Level_Manager();
_w1 := SEL(pump.Mode.eMode=eAnalog_Pump_Modes.Auto, pump.HMI_Volume_Target, pump.PLC_Volume_Target);
pump.Live_Rate := SEL(Pump.Config.Follow_ENABLE, _w1, Pump.Calibration_Rate* (pump.Config.Follow_Rate/100));
lcl_Target := _w1;
lcl_Seconds := SEL(pump.Mode.eMode=eAnalog_Pump_Modes.Auto, Pump.HMI_Volume_Target/PUMP.HMI_Rate_PCT, PUMP.PLC_Volume_Target/Pump.PLC_Rate_PCT);
_w2 := lcl_Target / ((PUMP.Config.Min_Speed/100.0) * (Pump.Calibration_Rate/60));
MAX_Time := _w2;
_w3 := lcl_Target / ((PUMP.Config.Max_Speed/100.0) * (Pump.Calibration_Rate/60));
Min_Time := _w3;
_w4 := SEL(lcl_Seconds<Min_time, SEL(lcl_Seconds>Max_Time, lcl_Seconds, _w2), _w3);
_w5 := REAL_TO_INT(_w4);
lcl_Seconds := _w5;
New_Pump_Time := _w5;
Base_PCT := SEL(lcl_Target=0, (Min_Time / _w4) * PUMP.Config.Max_Speed, 0.0);
_w6 := (Pump.Mode.eMode=eAnalog_Pump_Modes.Manual) OR Pump.PLC_Run AND (pump.Mode.eMode=eAnalog_Pump_Modes.Auto);
RUN_REQ := _w6;
_w7 := INT_TO_TIME(PUMP.Config.SuckBack_Seconds) * 1000;
_w8 := INT_TO_Time(New_Pump_Time) * 1000;
TON_0(IN := _w6, PT := _w8); // TON
_w9 := Pump.PLC_Run AND (pump.Mode.eMode=eAnalog_Pump_Modes.Auto);
_w10 := _w6 AND NOT TON_0.Q AND NOT (lcl_Target=0) OR (pump.Mode.eMode=eAnalog_Pump_Modes.Prime) OR (pump.Mode.eMode=eAnalog_Pump_Modes.Calibrate) OR Pump.Config.Follow_ENABLE;
F_TRIG_2(CLK := _w10); // F_Trig
Pump.Pump_FWD := _w10;
TP_2(IN := F_TRIG_2.Q AND (PUMP.Config.SuckBack_Seconds>1), PT := t#3s); // TP
TON_1(IN := TP_2.Q, PT := T#2s); // TON
TP_0(IN := TON_1.Q, PT := _w7); // TP
Pump.Pump_REV := TP_0.Q;
RUN := _w10 OR TP_0.Q;
REV := TP_0.Q;
PUMP.Batch_ETA := SEL(lcl_Target=0, SEL(_w6, New_Pump_time, TIME_TO_INT((_w8 - TON_0.ET) / 1000)), 0);
Pump.PCT_Remain := SEL(Run_REQ, 0.0, (1 - Pump.Volume_Delivered / pump.Live_Rate) * 100);
F_TRIG_0(CLK := _w9); // F_trig
IF F_TRIG_0.Q THEN _w11 := 0; END_IF
lcl_Target := _w11;
R_TRIG_0(CLK := Pump.Pump_FWD); // R_trig
Pump.Volume_Delivered := SEL(R_TRIG_0.Q, ((Pump.Calibration_Rate/60) * (Base_PCT/100)) * TIME_TO_INT(TON_0.ET / 1000), 0.0);
SET_Status();
F_TRIG_1(CLK := pump.Mode.eMode=eAnalog_Pump_Modes.Calibrate); // F_trig
_w12 := SEL(REV, 0, Pump.Config.SuckBack_Speed);
_w13 := (pump.HMI_Volume_Target / ((Pump.HMI_Volume_Target/ Pump.HMI_Rate_PCT) / 60.0)) * (100 / (pump.Config.Max_Speed*0.75));
Cal_Value := _w13;
IF F_TRIG_1.Q AND NOT TP_1.Q THEN _w14 := _w13; END_IF
Pump.Calibration_Rate := _w14;
_w15 := SEL(Pump.Pump_FWD, _w12, SEL(Pump.Config.Follow_ENABLE, SEL(pump.Mode.eMode=eAnalog_Pump_Modes.Prime, SEL(pump.Mode.eMode=eAnalog_Pump_Modes.Calibrate, Base_PCT, pump.Config.Max_Speed*0.75), pump.Config.Max_Speed), Pump.Config.Follow_Rate));
Pump.Pump_CV := _w15;
Speed := _w15;

ACTION Set_Status:
Pump.Status.eStatus := SEL((Pump.Mode.eMode=eAnalog_Pump_Modes.Auto) AND NOT Pump.PUMP_FWD AND PUMP.PLC_Run, SEL((Pump.Mode.eMode=eAnalog_Pump_Modes.Auto) AND Pump.Pump_FWD AND Pump.PLC_Run, SEL(Pump.Mode.eMode=eAnalog_Pump_Modes.Manual, SEL(Pump.Mode.eMode=eAnalog_Pump_Modes.Disabled, eAnalog_Pump_Status.IDLE, eAnalog_Pump_Status.Disabled), eAnalog_Pump_Status.Manual), eAnalog_Pump_Status.Running), eAnalog_Pump_Status.Complete);
END_ACTION

END_FUNCTION_BLOCK

// Level_2_Controls/Condensate_Trap_UDFB
FUNCTION_BLOCK Condensate_Trap_UDFB
VAR_INPUT
	LSHH:Burkert.DI_DUT;
	LSH:Burkert.DI_DUT;
	LSL:Burkert.DI_DUT;
	LSLL:Burkert.DI_DUT;
	Valve_Ready:BOOL;
	Steam_Load:REAL:=0;
	Purge_Duration:TIME:=T#15S;
	V2:BOOL:=FALSE;
	
END_VAR
VAR_OUTPUT
	ACV:REAL;
END_VAR

VAR
	R_TRIG_0: R_Trig;
	Valve_Min: REAL;
	Valve_Max: REAL;
	TON_0: TON;
	TON_2: TON;
	
	Target_CMD:REAL;
	T_mid:REAL;
	old_T_mid:REAL;
	t_Ramp:REAL:=0;
	Ramp: RAMP_REAL;
	Static_Time:Ton;
	Purge_TP:TP;
	purgeCount:UINT:=0;
	PurgeCount_rTrig:r_Trig;
END_VAR
VAR_IN_OUT
	Trap:cCondensate_Trap;
END_VAR
VAR // added by the converter: edge detectors and wires of the graphical bodies
    _w1, _w2, _w5, _w6, _w7, _w8, _w9, _w10, _w11, _w12, _w13, _w16, _w17, _w18 : ANY;
    _w3, _w4, _w14 : BOOL;
    _w15 : REAL;
END_VAR

_w1 := (LSL.Status.eStatus=Di_Status.Liquid_Detected) OR (LSL.Status.eStatus=Di_Status.Liquid_Detected_Alarm);
_w2 := (LSH.Status.eStatus=Di_Status.Liquid_Detected) OR (LSH.Status.eStatus=Di_Status.Liquid_Detected_Alarm);
_w3 := True;
IF _w3 THEN Positions(); END_IF
_w4 := _w3;
IF _w4 THEN Purge(); END_IF
IF _w4 THEN Status(); END_IF
_w5 := (LSHH.Status.eStatus=Di_Status.Liquid_Detected_Alarm) OR (LSHH.Status.eStatus=Di_Status.Liquid_Detected);
_w6 := (LSLL.Status.eStatus=Di_Status.Liquid_Detected) OR (LSLL.Status.eStatus=Di_Status.Liquid_Detected_Alarm);
_w7 := _w1 AND _w6;
IF TON_0.Q THEN _w8 := ACV+1; END_IF
_w9 := SEL(_w6, 100, Trap.Min_Valve_Positions[1]);
Trap.READY := Valve_Ready;
_w10 := _w2 AND _w7;
_w11 := _w5 AND _w10;
_w12 := SEL(_w11, SEL(_w10, SEL(_w7, _w9, Trap.Min_Valve_Positions[2]), Trap.Min_Valve_Positions[3]), 100);
_w13 := SEL(_w11, SEL(_w10, SEL(_w7, SEL(_w6, 0, Trap.Min_Valve_Positions[0]), Trap.Min_Valve_Positions[1]), Trap.Min_Valve_Positions[2]), Trap.Min_Valve_Positions[3]);
_w14 := _w13 <= 1;
TON_0(IN := NOT _w14 AND NOT TON_0.Q, PT := T#1s); // TON
_w15 := SEL(V2, SEL(_w14, LIMIT(_w13, _w8, _w12), 0.0), Target_CMD);
ACV := _w15;
Trap.CV := _w15;

ACTION Positions:


CASE Trap.Status OF
	eCondensate_Status.IDLE:
		Valve_Min:=0;
		Valve_Max:=0.1;
	eCondensate_Status.Stage_1:
		Valve_Min:=0;
		Valve_Max:=Trap.Min_Valve_Positions[0];
	eCondensate_Status.Stage_2:
		Valve_Min:=Trap.Min_Valve_Positions[0];
		Valve_Max:=Trap.Min_Valve_Positions[1];
	eCondensate_Status.High_Warning:
		Valve_Min:=Trap.Min_Valve_Positions[1];
		Valve_Max:=Trap.Min_Valve_Positions[2];
	eCondensate_Status.Fault:
		Valve_Min:=Trap.Min_Valve_Positions[2];
		Valve_Max:=Trap.Min_Valve_Positions[3];
		
		eCondensate_Status.HIGH_Alarm:
		Valve_Min:=Trap.Min_Valve_Positions[2];
		Valve_Max:=Trap.Min_Valve_Positions[3];
		
	eCondensate_Status.Level_Switch_Fault:
		Valve_Min:=0;
		Valve_Max:=0.1;
			
	eCondensate_Status.Purge:
		Valve_Min:=Trap.Min_Valve_Positions[1];
		Valve_Max:=Trap.Min_Valve_Positions[1]+1;
		Trap.PLC_Purge:=FALSE;
		IF Trap.Purge.eMode=Burkert.eHOA_Modes.Manual THEN Trap.Purge.eMode:=Burkert.eHOA_Modes.Auto; END_IF;
	
END_CASE

t_mid:=fbMidPoint(High:=Valve_max,Low:=Valve_Min);
Static_Time(PT:=T#2M, 
	IN:= (	t_mid = Old_t_mid AND 
			Trap.CV<15 AND
			Steam_Load>75)
	);
	
IF t_mid > Old_t_mid THEN
	t_Ramp:=Valve_Max;
	Old_T_Mid:=t_Mid;
END_IF;

IF t_mid < Old_t_mid THEN
	t_Ramp:=Valve_Min;
	Old_T_Mid:=t_Mid;
END_IF;



Ramp(
	IN:= t_ramp, 
	ASCEND:= 2, 
	DESCEND:= 2, 
	TIMEBASE:= T#1S, 
	RESET:= FALSE );

IF Ramp.OUT<5  THEN
	Target_CMD:=0;
ELSE
	Target_CMD:=LIMIT (Valve_Min,Ramp.OUT,MIN(Valve_Max,100));
END_IF
END_ACTION

ACTION Purge:
Purge_TP(PT:=Purge_Duration);




CASE Trap.Purge.eMode OF
	Burkert.eHOA_Modes.Off:
		Purge_TP.IN:=FALSE;
	Burkert.eHOA_Modes.Manual:
		Purge_TP.IN:=TRUE;
	Burkert.eHOA_Modes.Auto:
		Purge_TP.IN:=Static_Time.Q OR Trap.PLC_Purge;
		Trap.PLC_Purge:=FALSE;
END_CASE

PurgeCount_rTrig(CLK:=Purge_TP.IN);
IF PurgeCount_rTrig.Q THEN PurgeCount:=PurgeCount+1;	END_IF;
END_ACTION

ACTION Status:
TON_2(IN := ACV>99, PT := T#30s); // TON
_w16 := (LSLL.Status.eStatus=Di_Status.Liquid_Detected) OR (LSLL.Status.eStatus=Di_Status.Liquid_Detected_Alarm);
_w17 := ((LSL.Status.eStatus=Di_Status.Liquid_Detected) OR (LSL.Status.eStatus=Di_Status.Liquid_Detected_Alarm)) AND _w16;
_w18 := ((LSH.Status.eStatus=Di_Status.Liquid_Detected) OR (LSH.Status.eStatus=Di_Status.Liquid_Detected_Alarm)) AND _w17;
Trap.Status := SEL(Purge_TP.Q AND NOT (Trap.Purge.eMode=Burkert.eHOA_Modes.Off), SEL(LSHH.Raw AND NOT LSH.Raw OR LSH.Raw AND NOT LSL.Raw OR LSL.Raw AND NOT LSLL.Raw, SEL(TON_2.Q, SEL(((LSHH.Status.eStatus=Di_Status.Liquid_Detected_Alarm) OR (LSHH.Status.eStatus=Di_Status.Liquid_Detected)) AND _w18, SEL(_w18, SEL(_w17, SEL(_w16, eCondensate_Status.IDLE, eCondensate_Status.Stage_1), eCondensate_Status.Stage_2), eCondensate_Status.High_Warning), eCondensate_Status.HIGH_Alarm), eCondensate_Status.Fault), eCondensate_Status.Level_Switch_Fault), eCondensate_Status.Purge);
END_ACTION

END_FUNCTION_BLOCK

// Level_2_Controls/DofMaster
FUNCTION_BLOCK DofMaster
VAR_INPUT
	Config:REFERENCE TO cDOF_Master;
	ALL_Lines_Ready:BOOL;
	
END_VAR
VAR_OUTPUT
END_VAR
VAR
	R_Trig_0:R_trig;
	Batch_CLK:TON;
	R_Trig_1:R_trig;
	
END_VAR

Config.StrBatch_Mode:=Burkert_OSCAT_BASIC.REPLACE_ALL(str:=TO_STRING(Config.Batch_Mode.eMode), src:='_' , rep:=' ' );
Config.StrBatch_Status:=Burkert_OSCAT_BASIC.REPLACE_ALL(str:=TO_STRING(Config.Batch_Status.eStatus), src:='_' , rep:=' ' );
Config.StrBatch_Task:= Burkert_OSCAT_BASIC.REPLACE_ALL(str:=TO_STRING(Config.Batch_Task.eTask), src:='_' , rep:=' ' );

Config.Batch_Target_ms:=TO_UDINT((Config.Batch_Volume/Config.Batch_Rate)*60*1000);
Config.Batch_Elapsed_ms:=TO_UDINT(Batch_CLK.ET);
Config.Batch_Remain_ms:=Config.Batch_Target_ms-Config.Batch_Elapsed_ms;

R_trig_1( CLK:=(Config.Batch_Mode.eMode=Burkert.eHOA_Modes.Manual));

Batch_CLK(IN:=Config.Batch_Task.eTask=eBatch_Task.Run,PT:=T#6H);
Config.Batch_CLK:=Batch_CLK.ET;

IF Config.Current_Batch_Rate >0 THEN
	Config.Batch_ETA_ms:=TO_UDINT(	((Config.Batch_Volume-Config.Current_Batch_Volume) / Config.Current_Batch_Rate)*(60*1000)	);
ELSE
	Config.Batch_ETA_ms:=0;
END_IF;

IF Config.Batch_Rate >0 THEN	
	Config.Batch_Target_ms:=TO_UDINT((Config.Batch_Volume/Config.Batch_Rate)*60*1000);
	Config.Batch_Remain:=TO_TIME(		(Config.Batch_Volume/Config.Batch_Rate)*60*1000)-Config.Batch_CLK;
ELSE
	Config.Batch_Remain:=T#0MS;
	Config.Batch_Target_ms:=0;
END_IF


IF Config.Batch_Volume>0 THEN
	Config.Current_Batch_PCT:=(Config.Current_Batch_Volume/Config.Batch_Volume)*100;
ELSE
	Config.Current_Batch_PCT:=0;
	Config.Batch_Status.eStatus:=eBatch_Status.Idle;
END_IF;


IF ALL_Lines_Ready THEN
	Config.Batch_Status.eStatus:=eBatch_Status.Ready;
	IF Config.Batch_Task.eTask=eBatch_task.Resume THEN Task_resume(); END_IF;
	IF Config.Current_Batch_Rate>0.5 THEN Config.Batch_Status.eStatus:=eBatch_Status.Active; END_IF;
	
	CASE Config.Batch_Mode.eMode OF
		Burkert.eHOA_Modes.Auto:
			IF Config.PLC_Run THEN 
				Config.Batch_Task.eTask:=eBatch_Task.Run; 
			ELSE
				Config.Batch_Task.eTask:=eBatch_Task.OFF;
			END_IF;
		Burkert.eHOA_Modes.Manual:  
			IF R_trig_1.q	THEN	Config.Batch_Task.eTask:=eBatch_Task.Run; END_IF;
	ELSE
		Config.Batch_Task.eTask:=eBatch_Task.OFF;
		Config.Batch_Status.eStatus:=eBatch_Status.Disabled;
		Config.PLC_Run:=FALSE;
	END_CASE
ELSE
	Config.Batch_Task.eTask:=eBatch_Task.OFF;
	Config.Batch_Status.eStatus:=eBatch_Status.Fault;
	Config.Batch_Mode.eMode:=Burkert.eHOA_Modes.Off;
END_IF;

IF Config.Current_Batch_PCT>=100.0 THEN Config.Batch_Status.eStatus:=eBatch_Status.Complete; END_IF;


R_Trig_0(CLK:=Config.Batch_Task.eTask=eBatch_task.Run);
IF R_Trig_0.Q THEN
	Config.MasterID:=Config.MasterID+1;
END_IF;

END_FUNCTION_BLOCK

// Level_2_Controls/Duplex_VFD
FUNCTION_BLOCK Duplex_VFD
VAR_INPUT
	VFD1:REFERENCE TO Burkert.VFD_Control;
	VFD2:REFERENCE TO Burkert.VFD_Control;
	
END_VAR
VAR_OUTPUT
END_VAR
VAR
	VFD1_Primary:BOOL;
END_VAR

VAR_IN_OUT
	Duplex:cDuplex;
END_VAR
VAR // added by the converter: edge detectors and wires of the graphical bodies
    _w1 : ANY;
    _w2, _w3 : BOOL;
END_VAR

IF NOT(VFD2.RunTime_Minutes=0) THEN	
	Duplex.Current_Split := TO_REAL(VFD1.RunTime_Minutes/VFD2.RunTime_Minutes)*100;
END_IF;
IF VFD1.Actual=0 AND VFD2.Actual=0 AND Duplex.Run_Request=FALSE THEN
	VFD1_Primary:=Duplex.Current_Split<Duplex.Target_Split;
END_IF

Outputs();

ACTION Outputs:
_w1 := NOT VFD1.Ready AND VFD2.Ready;
_w2 := SEL(VFD1_Primary AND VFD1.Ready OR VFD1.Ready AND NOT VFD2.Ready, False, Duplex.Run_request);
VFD1.PLC_CMD := SEL(_w2, 0.0, Duplex.Run_PCT);
VFD1.PLC_Run := _w2;
_w3 := SEL(NOT VFD1_Primary AND VFD2.Ready OR _w1, False, Duplex.Run_Request);
VFD2.PLC_Run := _w3;
VFD1.PLC_CMD := SEL(_w3, 0.0, Duplex.Run_PCT);
END_ACTION

END_FUNCTION_BLOCK

// Level_2_Controls/PID_UDFB
FUNCTION_BLOCK PID_UDFB
VAR_INPUT
	Reverse:BOOL;
	CV_OK:BOOL;
	PV_OK:BOOL;
END_VAR
VAR_OUTPUT
	CV:REAL;
END_VAR
VAR
	FT_PIDW_0: BURKERT_OSCAT_BASIC.FT_PIDW;
	R_TRIG_0: R_trig;
	Loop_Enable: BOOL;
	R_TRIG_1: R_Trig;
END_VAR
VAR_IN_OUT
	PID:cPID_DUT;
END_VAR
VAR // added by the converter: edge detectors and wires of the graphical bodies
    _w1, _w2, _w3, _w4, _w6, _w7 : ANY;
    _w5 : BOOL;
END_VAR

PID_Status();
R_TRIG_0(CLK := PID.MODE.eMode=ePID_Modes.Auto); // R_trig
IF R_TRIG_0.Q THEN _w1 := PID.HMI_Target; END_IF
PID.PLC_Target := _w1;
_w2 := SEL(PID.MODE.eMode=ePID_Modes.Auto, PId.HMI_Target, PID.PLC_Target);
PID.Live_Target := _w2;
_w3 := _w2 * PID.FF;
PID.CV_FF := _w3;
_w4 := SEL(Reverse, _w2 - PID.Actual, PID.Actual - _w2);
PID.Err := _w4;
_w5 := SEL(PID.MODE.eMode=ePID_Modes.Auto, PID.MODE.eMode=ePID_Modes.FORCED_ON, PID.PLC_Enable AND (Not(PID.Inhibit))) AND True AND CV_OK AND PV_OK;
Loop_Enable := _w5;
FT_PIDW_0(
    IN := _w4,
    KP := PID.KP,
    TN := PID.TN,
    TV := PID.TV,
    LIM_L := PID.CV_Min-PID.CV_FF,
    LIM_H := PID.CV_Max-PID.CV_FF,
    RST := R_Trig_1.Q OR NOT _w5); // BURKERT_OSCAT_BASIC.FT_PIDW
_w6 := SEL(Loop_Enable, PID.CV_Min, _w3 + FT_PIDW_0.Y);
CV := _w6;
PID.CV := _w6;
PID.CV_P := PID.Err * PID.KP;
PID.CV_I := FT_PIDW_0.YI;
PID.CV_D := FT_PIDW_0.diff.out;
PID.Ready := (PID.MODE.eMode=ePID_Modes.Auto) AND CV_OK AND PV_OK;
R_TRIG_1(CLK := (PID.CV_P>0) AND (PID.CV_I<0) AND (FT_PIDW_0.Y<0.5) AND _w5); // R_Trig
IF NOT (PID.MODE.eMode=ePID_Modes.FORCED_ON) THEN _w7 := PID.PLC_Target; END_IF
PID.HMI_Target := _w7;

END_FUNCTION_BLOCK

// Level_2_Controls/Quick_Mix_UDFB
FUNCTION_BLOCK Quick_Mix_UDFB
VAR_INPUT
	Destination_OK:BOOL;
END_VAR
VAR_OUTPUT
	//Active:BOOL;
	OK:BOOL;
END_VAR
VAR
	Current_Mode:eQuick_Mix_modes;
	Current_Status:eQuick_Mix_Status;
	SFCReset:BOOL;
	SFCInit:BOOL;
	PLC_Active:BOOL;
	Temp_PID:BURKERT_OSCAT_BASIC.FT_PIDW;
	Flow_PID:BURKERT_OSCAT_BASIC.FT_PIDW;
	Ramp:Burkert_OSCAT_BASIC.SRAMP;
	tRamp:Burkert_OSCAT_BASIC.SRAMP;
	Ramp_Time:TIME;
	Pause_Active:BOOL;
	Pause_Ton:Ton;
	//Temp_Control:Burkert_OSCAT_BASIC.SCALE_R;
	//Flow_Control:Burkert_OSCAT_BASIC.SCALE_R;
	tHW:REAL;
END_VAR
VAR_IN_OUT
	HW		:Burkert.cACV;
	CW		:Burkert.cACV;
	FIT		:Burkert.cFIT;
	TT		:Burkert.cSensor;
	Loop	:Quick_Mix_Dut;
END_VAR

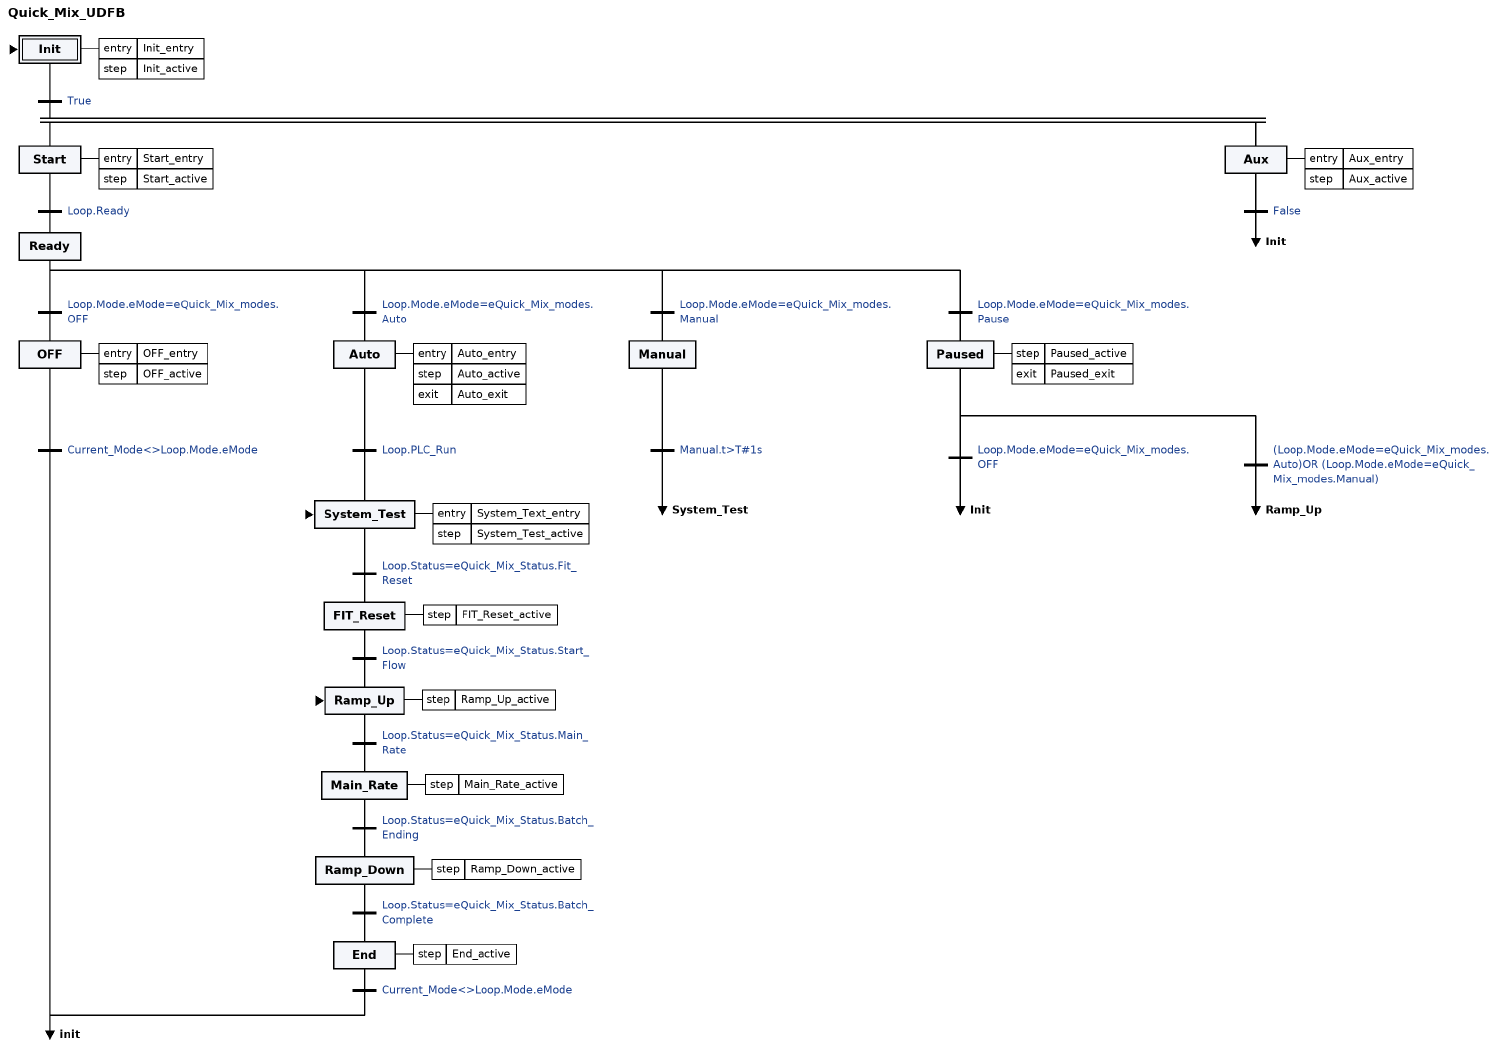
INITIAL_STEP Init:
    Init_entry(P1);  // entry action
    Init_active(N);  // step action
END_STEP
TRANSITION FROM Init TO (Start, Aux)
    := True;
END_TRANSITION
STEP Start:
    Start_entry(P1);  // entry action
    Start_active(N);  // step action
END_STEP
TRANSITION FROM Start TO Ready
    := Loop.Ready;
END_TRANSITION
STEP Ready:
END_STEP
STEP Aux:
    Aux_entry(P1);  // entry action
    Aux_active(N);  // step action
END_STEP
TRANSITION FROM Aux TO Init
    := False;
END_TRANSITION
TRANSITION FROM Ready TO OFF
    := Loop.Mode.eMode=eQuick_Mix_modes.OFF;
END_TRANSITION
STEP OFF:
    OFF_entry(P1);  // entry action
    OFF_active(N);  // step action
END_STEP
TRANSITION FROM OFF TO init
    := Current_Mode<>Loop.Mode.eMode;
END_TRANSITION
TRANSITION FROM Ready TO Auto
    := Loop.Mode.eMode=eQuick_Mix_modes.Auto;
END_TRANSITION
STEP Auto:
    Auto_entry(P1);  // entry action
    Auto_active(N);  // step action
    Auto_exit(P0);  // exit action
END_STEP
TRANSITION FROM Auto TO System_Test
    := Loop.PLC_Run;
END_TRANSITION
STEP System_Test:
    System_Text_entry(P1);  // entry action
    System_Test_active(N);  // step action
END_STEP
TRANSITION FROM System_Test TO FIT_Reset
    := Loop.Status=eQuick_Mix_Status.Fit_Reset;
END_TRANSITION
STEP FIT_Reset:
    FIT_Reset_active(N);  // step action
END_STEP
TRANSITION FROM FIT_Reset TO Ramp_Up
    := Loop.Status=eQuick_Mix_Status.Start_Flow;
END_TRANSITION
STEP Ramp_Up:
    Ramp_Up_active(N);  // step action
END_STEP
TRANSITION FROM Ramp_Up TO Main_Rate
    := Loop.Status=eQuick_Mix_Status.Main_Rate;
END_TRANSITION
STEP Main_Rate:
    Main_Rate_active(N);  // step action
END_STEP
TRANSITION FROM Main_Rate TO Ramp_Down
    := Loop.Status=eQuick_Mix_Status.Batch_Ending;
END_TRANSITION
STEP Ramp_Down:
    Ramp_Down_active(N);  // step action
END_STEP
TRANSITION FROM Ramp_Down TO End
    := Loop.Status=eQuick_Mix_Status.Batch_Complete;
END_TRANSITION
STEP End:
    End_active(N);  // step action
END_STEP
TRANSITION FROM End TO init
    := Current_Mode<>Loop.Mode.eMode;
END_TRANSITION
TRANSITION FROM Ready TO Manual
    := Loop.Mode.eMode=eQuick_Mix_modes.Manual;
END_TRANSITION
STEP Manual:
END_STEP
TRANSITION FROM Manual TO System_Test
    := Manual.t>T#1s;
END_TRANSITION
TRANSITION FROM Ready TO Paused
    := Loop.Mode.eMode=eQuick_Mix_modes.Pause;
END_TRANSITION
STEP Paused:
    Paused_active(N);  // step action
    Paused_exit(P0);  // exit action
END_STEP
TRANSITION FROM Paused TO Init
    := Loop.Mode.eMode=eQuick_Mix_modes.OFF;
END_TRANSITION
TRANSITION FROM Paused TO Ramp_Up
    := (Loop.Mode.eMode=eQuick_Mix_modes.Auto)OR (Loop.Mode.eMode=eQuick_Mix_modes.Manual);
END_TRANSITION

ACTION Auto_active:
//Flow_PiD(RST:=TRUE);
Flow_PID.PLC_Enable:=FALSE;
Temp_PID(RST:=TRUE);
Loop.Actual_Rate:=0;
Ramp.X:=0;

Loop.Live_Rate:=Ramp.Y;
tRamp.X:=TT.EU;	

Loop.Live_Temp:=tRamp.Y;
Loop.Status:=eQuick_Mix_Status.IDLE;
Loop.Active:=FALSE;
END_ACTION

ACTION Aux_active:
IF Current_Mode<>Loop.Mode.eMode AND NOT(Pause_Active)THEN
	Current_Mode:=Loop.Mode.eMode;
	SFCReset:=TRUE;
END_IF

IF PLC_Active AND NOT(Loop.PLC_Run) OR (FIT.Rate.EU>10 AND FIT.Total>Loop.Target_Volume+15) THEN
	PLC_Active:=FALSE;
	SFCReset:=TRUE;
	Flow_PID.PLC_Enable:=FALSE;
	loop.Status:=eQuick_Mix_Status.Batch_Complete;
END_IF;

IF LOOP.Active AND (FIT.Rate.EU>10 AND FIT.Total>Loop.Target_Volume+15) THEN
	PLC_Active:=FALSE;
	Flow_PID.PLC_Enable:=FALSE;
	loop.Status:=eQuick_Mix_Status.Batch_Complete;
END_IF;



	
Current_Status:=Loop.Status;
Loop.Actual_Temp:=TT.EU;


IF LOOP.Active THEN
	Loop.Actual_Rate:=FIT.Rate.EU;
	Loop.Actual_Volume:=FIT.Total;
END_IF




IF FIT.Rate.EU > 1 AND Loop.Active THEN
	Loop.ETA:= TO_UDINT((((loop.Target_Volume-Loop.Actual_Volume)/FIT.Rate.EU)*60.0)-TO_INT(Ramp_Time/2000))*1000 ;
	Loop.PCT_Complete:= ((FIT.Total/Loop.Target_Volume)*100);
	Loop.PCT_Remain:=100.0-Loop.PCT_Complete;
ELSE
	//Loop.ETA:=0;
	//Loop.PCT_Complete:=100;
	//Loop.PCT_Remain:=0;
END_IF;

Pause_Ton(PT:=T#10S,IN:=(HW.PLC_CMD	> 5 OR  CW.PLC_CMD>5) AND NOT(Destination_OK) AND Loop.Active);
IF  Pause_TON.Q THEN
	Loop.Mode.eMode	:=eQuick_Mix_modes.Pause;
	Pause_Active:=TRUE;
END_IF;


Loop.Temp_Control:=Burkert_OSCAT_BASIC.SCALE_R(
	X:=TT.EU , 
	I_LO:= Loop.Target_Temp-(Loop.Config.Temp_Window_Alarm*2), 
	I_HI:= Loop.Target_Temp+(Loop.Config.Temp_Window_Alarm*2), 
	O_LO:= 0, 
	O_HI:=100 );
//Burkert_OSCAT_BASIC.SCALE_R.SCALE_R;


Loop.Flow_Control:=Burkert_OSCAT_BASIC.SCALE_R(
	X:=FIT.Rate.EU , 
	I_LO:= Loop.Target_Rate-(Loop.Config.Flow_Window_Alarm*2), 
	I_HI:= Loop.Target_Rate+(Loop.Config.Flow_Window_Alarm*2), 
	O_LO:= 0, 
	O_HI:=100 );
//Loop.Flow_Control:=Burkert_OSCAT_BASIC.SCALE_R.SCALE_R;
Loop.HW_Valve:=HW.Valve_Actual;
Loop.CW_Valve:=CW.Valve_Actual;
Loop.Temp_CV:=Temp_PID.Y;
Loop.Flow_CV:=Flow_PID.CV;
IF NOT(loop.PLC_Run) THEN
		Loop.Status:=eQuick_mix_Status.IDLE;
END_IF;
Loop.Ready:=(HW.Ready AND CW.Ready AND TT.Ready);

IF NOT(HW.Ready) THEN	Loop.Status:=eQuick_mix_Status.HW_Valve_Not_Ready;	END_IF;

IF NOT(CW.Ready) THEN	Loop.Status:=eQuick_mix_Status.CW_Valve_Not_Ready;	END_IF;

IF NOT(TT.Ready) THEN	Loop.Status:=eQuick_mix_Status.TT_Not_Ready;	END_IF;


Flow_PID.CV_Min:=0;
Flow_PID.CV_Max:=100;

Flow_PID.KP:=Loop.Config.Flow_KP;
FLow_PID.TN:=Loop.Config.Flow_TN;
Flow_PID.TV:=Loop.Config.Flow_TV;

//tt.Alarm_Config.Setpoints.Target:=Loop.Target_Temp;
TT.Alarm_Config.Setpoints.Hysteresis:=0.5;
TT.Alarm_Config.Setpoints.Hi_Norm:=TT.Alarm_Config.Setpoints.Hi_Warn-1;
TT.Alarm_Config.Setpoints.Low_Norm:=TT.Alarm_Config.Setpoints.Low_warn+1;
TT.Alarm_Config.Setpoints.Warn_Debounce:=5;





Ramp(
	A_UP:=Loop.Config.Ramp_Rate,
	A_DN:=0-Loop.Config.Ramp_Rate,
	VU_Max:=50,
	VD_Max:=-50,
	Limit_High:=Loop.Target_Rate+0.1,
	Limit_Low:=MIN(Loop.Config.Min_Flow, Loop.Target_Rate)-0.1,
	RST:=FALSE
);
	
tRamp(
	A_UP:=1,
	A_DN:=(-1),
	VU_Max:=50,
	VD_Max:=-50,
	Limit_High:=100,
	Limit_Low:=0,
	RST:=FALSE
);
END_ACTION

ACTION End_active:
CW.PLC_CMD:=0;
HW.PLC_CMD:=0;
Loop.Active:=FALSE;
Flow_PID.PLC_Enable:=FALSE;

////Flow_PID.PLC_Enable:=(End_Active.tT
END_ACTION

ACTION FIT_Reset_active:
Flow_PiD(RST:=TRUE);
Temp_PID(RST:=TRUE);

TT.Alarm_Config.Setpoints.Alarm_Debounce	:=loop.Config.Alarm_Debounce;
TT.Alarm_Config.Setpoints.Hi_Warn:=( loop.Target_Temp+ loop.Config.Temp_WIndow_Warn);
TT.Alarm_Config.Setpoints.Low_Warn:=( loop.Target_Temp- loop.Config.Temp_WIndow_Warn);
TT.Alarm_Config.Setpoints.Hi_Hi_Alarm:=(Loop.Target_Temp+Loop.Config.Temp_Window_Alarm);
TT.Alarm_Config.Setpoints.Low_Low_Alarm:=(Loop.Target_Temp-Loop.Config.Temp_Window_Alarm);
TT.Alarm_Config.Silence:=TRUE;

FIT.Rate.Alarm_Config.Setpoints.Alarm_Debounce	:=loop.Config.Alarm_Debounce;
FIT.Rate.Alarm_Config.Setpoints.Hi_Warn:=( FIT.Rate.EU+ loop.Config.Flow_WIndow_Warn);
FIT.Rate.Alarm_Config.Setpoints.Low_Warn:=( FIT.Rate.EU- loop.Config.Flow_WIndow_Warn);
FIT.Rate.Alarm_Config.Setpoints.Hi_Hi_Alarm:=(FIT.Rate.EU+Loop.Config.Flow_Window_Alarm);
FIT.Rate.Alarm_Config.Setpoints.Low_Low_Alarm:=(FIT.Rate.EU-Loop.Config.Flow_Window_Alarm);
FIT.Rate.Alarm_Config.Silence:=TRUE;


Flow_PID.KP:=Loop.Config.Flow_KP;
Flow_PID.TN:=Loop.Config.Flow_TN;
Flow_PID.TV:=Loop.Config.Flow_TV;
Flow_PID.LIM_H:=100;
Flow_PID.LIM_L:=0;


Temp_PID.KP:=Loop.Config.Temp_KP;
Temp_PID.TN:=Loop.Config.Temp_TN;
Temp_PID.TV:=Loop.Config.Temp_TV;
Temp_PID.LIM_H:=100;
Temp_PID.LIM_L:=-100;


FIT.PLC_Reset:=(FIT.Total>1);

IF (FIT.Total<1) THEN
	Loop.Status:=eQuick_Mix_Status.Start_Flow;
END_IF
Ramp(x:=0,
	A_UP:=Loop.Config.Ramp_Rate,
	A_DN:=0-Loop.Config.Ramp_Rate,
	VU_Max:=50,
	VD_Max:=-50,
	Limit_High:=500,
	Limit_Low:=Loop.Config.Min_Flow,
	RST:=TRUE);
	
tRamp(x:=TT.EU,
	A_UP:=1,
	A_DN:=(-1),
	VU_Max:=50,
	VD_Max:=-50,
	Limit_High:=100,
	Limit_Low:=0,
	RST:=FALSE);


TT.Alarm_Config.Setpoints.Alarm_Debounce	:=loop.Config.Alarm_Debounce;
TT.Alarm_Config.Setpoints.Hi_Warn:=( tRamp.Y+ loop.Config.Temp_WIndow_Warn);
TT.Alarm_Config.Setpoints.Low_Warn:=( tRamp.Y- loop.Config.Temp_WIndow_Warn);
TT.Alarm_Config.Setpoints.Hi_Hi_Alarm:=(tRamp.Y+Loop.Config.Temp_Window_Alarm);
TT.Alarm_Config.Setpoints.Low_Low_Alarm:=(tRamp.Y-Loop.Config.Temp_Window_Alarm);
END_ACTION

ACTION Init_active:
SFCReset:=FALSE;
SFCInit:=FALSE;

Flow_PID.PLC_Enable:=False;
END_ACTION

ACTION Init_entry:
SFCReset:=FALSE;
SFCInit:=FALSE;
Loop.Active:=FALSE;
Flow_PID.RST:=TRUE;
Temp_PID.RST:=TRUE;
CW.Mode.eMode:=Burkert.eACV_Modes.Auto;
HW.Mode.eMode:=Burkert.eACV_Modes.Auto;

CW.PLC_CMD:=0;
HW.PLC_CMD:=0;
OK:=FALSE;
Loop.Status:=eQuick_Mix_Status.IDLE;
Current_Mode:=Loop.Mode.eMode;
END_ACTION

ACTION Main_Rate_active:
Flow_PID.KP:=Loop.Config.Flow_KP;
Flow_PID.TN:=Loop.Config.Flow_TN;
Flow_PID.TV:=Loop.Config.Flow_TV;
Flow_pid.LIM_L:=0;
Flow_PID.LIM_H:=100;

Temp_PID.KP:=Loop.Config.Temp_KP;
Temp_PID.TN:=Loop.Config.Temp_TN;
Temp_PID.TV:=Loop.Config.Temp_TV;
Temp_pid.LIM_L:=(-100);
Temp_PID.LIM_H:=100;



Ramp(x:=Loop.Target_Rate, Rst:=FALSE);
Loop.Live_Rate:=Ramp.Y;
FIT.Rate.Alarm_Config.Setpoints.Alarm_Debounce	:=loop.Config.Alarm_Debounce;
FIT.Rate.Alarm_Config.Setpoints.Hi_Warn:=( Ramp.Y+ loop.Config.Flow_WIndow_Warn);
FIT.Rate.Alarm_Config.Setpoints.Low_Warn:=( Ramp.y- loop.Config.Flow_WIndow_Warn);
FIT.Rate.Alarm_Config.Setpoints.Hi_Hi_Alarm:=(Ramp.Y+Loop.Config.Flow_Window_Alarm);
FIT.Rate.Alarm_Config.Setpoints.Low_Low_Alarm:=(Ramp.Y-Loop.Config.Flow_Window_Alarm);
FIT.Rate.Alarm_Config.Silence:=FALSE;
Flow_PID(In:=Ramp.Y-FIT.Rate.EU,RST:=FALSE);

tRamp(x:=Loop.Target_Temp, Rst:=FALSE);
TT.Alarm_Config.Setpoints.Hi_Warn:=( tRamp.Y+ loop.Config.Temp_WIndow_Warn);
TT.Alarm_Config.Setpoints.Low_Warn:=( tRamp.Y- loop.Config.Temp_WIndow_Warn);
TT.Alarm_Config.Setpoints.Hi_Hi_Alarm:=(tRamp.Y+Loop.Config.Temp_Window_Alarm);
TT.Alarm_Config.Setpoints.Low_Low_Alarm:=(tRamp.Y-Loop.Config.Temp_Window_Alarm);
TT.Alarm_Config.Silence:=FALSE;
Loop.Live_Temp	:=tRamp.Y;
Temp_PID(In:=tRamp.Y-TT.EU,RST:=FALSE);


HW.PLC_CMD:= LIMIT(0, ((1+(Temp_PID.Y/100)) * Flow_PID.Y),100);
CW.PLC_CMD:= LIMIT(0, ((1-(Temp_PID.Y/100)) * Flow_PID.Y),100);
	
Loop.Active:=TRUE;





loop.Status:=eQuick_Mix_Status.On_Target;

IF TT.Status.eStatus=Burkert.eSensor_Status.High_Warning OR TT.Status.eStatus=Burkert.eSensor_Status.Low_Warning  THEN
	Loop.Status:=eQuick_Mix_Status.Temp_Warning;
END_IF;

IF TT.Status.eStatus=Burkert.eSensor_Status.HiHi_Alarm OR TT.Status.eStatus=Burkert.eSensor_Status.Low_Low_Alarm  THEN
	Loop.Status:=eQuick_Mix_Status.Temp_Fault;
	Loop.Mode.eMode:=eQuick_Mix_Modes.Pause;
END_IF;

IF FIT.Rate.Status.eStatus=Burkert.eSensor_Status.High_Warning OR FiT.Rate.Status.eStatus=Burkert.eSensor_Status.Low_Warning  THEN
	Loop.Status:=eQuick_Mix_Status.Flow_Warning;
END_IF;

IF FIT.Rate.Status.eStatus=Burkert.eSensor_Status.HiHi_Alarm OR FiT.Rate.Status.eStatus=Burkert.eSensor_Status.Low_Low_Alarm  THEN
	Loop.Status:=eQuick_Mix_Status.Flow_Fault;
	Loop.Mode.eMode:=eQuick_Mix_Modes.Pause;
END_IF;


OK:=(Loop.Status=eQuick_Mix_Status.On_Target);


IF Loop.ETA < 1 THEN
	Loop.Status:=eQuick_Mix_Status.Batch_Ending;
END_IF;
END_ACTION

ACTION OFF_active:
tRamp(x:=TT.Sensor.EU,
	A_UP:=1,
	A_DN:=(-1),
	VU_Max:=50,
	VD_Max:=-50,
	Limit_High:=100,
	Limit_Low:=0,
	RST:=FALSE);
Loop.Active:=FALSE;
Flow_PID(In:=0,RST:=TRUE);
Temp_PID(In:=0,RST:=TRUE);

HW.PLC_CMD:=0;
CW.PLC_CMD:=0;
Loop.Actual_Rate:=0;
END_ACTION

ACTION OFF_entry:
HW.PLC_CMD:=0;
CW.PLC_CMD:=0;
FIT.PLC_Reset:=FALSE;
Loop.Status:=eQuick_mix_Status.IDle;
Flow_PID.PLC_Enable:=FALSE;
Temp_PID(RST:=TRUE);
Loop.Active:=FALSE;
END_ACTION

ACTION Paused_active:
HW.PLC_CMD	:=0;
CW.PLC_CMD	:=0;
Loop.Flow_CV:=0;
Loop.Temp_CV:=0;
Temp_PID.RST:=TRUE;
Flow_PID.RST:=TRUE;
Loop.Actual_Rate:=0;


OK:=FALSE;
Loop.Active:=FALSE;
Pause_Active:=TRUE;
IF (Loop.Status <> eQuick_Mix_Status.Temperature_Fault) AND (Loop.Status <> eQuick_Mix_Status.Flow_Fault) THEN
	//Loop.Status:=eQuick_Mix_Status.Paused;
END_IF;




Ramp(x:=0,
	A_UP:=Loop.Config.Ramp_Rate,
	A_DN:=0-Loop.Config.Ramp_Rate,
	VU_Max:=50,
	VD_Max:=-50,
	Limit_High:=Loop.Target_Rate,
	Limit_Low:=Loop.Config.Min_Flow,
	RST:=FALSE);
Loop.Live_Rate:=Ramp.Y;
	
tRamp(x:=TT.Sensor.EU,
	A_UP:=1,
	A_DN:=(-1),
	VU_Max:=50,
	VD_Max:=-50,
	Limit_High:=100,
	Limit_Low:=0,
	RST:=FALSE);
Loop.Live_Temp:=tRamp.Y;
END_ACTION

ACTION Ramp_Down_active:
Flow_PID.KP:=Loop.Config.Flow_KP;
Flow_PID.TN:=Loop.Config.Flow_TN;
Flow_PID.TV:=Loop.Config.Flow_TV;
Flow_pid.LIM_L:=0;
Flow_PID.LIM_H:=100;

Temp_PID.KP:=Loop.Config.Temp_KP;
Temp_PID.TN:=Loop.Config.Temp_TN;
Temp_PID.TV:=Loop.Config.Temp_TV;
Temp_pid.LIM_L:=(-100);
Temp_PID.LIM_H:=100;



Loop.Status:=eQuick_Mix_Status.Batch_Ending;

Ramp(x:=Loop.Config.Min_Flow, Rst:=FALSE);
FIT.Rate.Alarm_Config.Setpoints.Alarm_Debounce	:=loop.Config.Alarm_Debounce;
FIT.Rate.Alarm_Config.Setpoints.Hi_Warn:=( Ramp.Y+ loop.Config.Flow_WIndow_Warn);
FIT.Rate.Alarm_Config.Setpoints.Low_Warn:=( Ramp.y- loop.Config.Flow_WIndow_Warn);
FIT.Rate.Alarm_Config.Setpoints.Hi_Hi_Alarm:=(Ramp.Y+Loop.Config.Flow_Window_Alarm);
FIT.Rate.Alarm_Config.Setpoints.Low_Low_Alarm:=(Ramp.Y-Loop.Config.Flow_Window_Alarm);
Loop.Live_Rate:=Ramp.Y;
Flow_PID(In:=Ramp.Y-FIT.Rate.EU,RST:=FALSE);

tRamp(x:=Loop.Target_Temp, Rst:=FALSE);
TT.Alarm_Config.Setpoints.Hi_Warn:=( tRamp.Y+ loop.Config.Temp_WIndow_Warn);
TT.Alarm_Config.Setpoints.Low_Warn:=( tRamp.Y- loop.Config.Temp_WIndow_Warn);
TT.Alarm_Config.Setpoints.Hi_Hi_Alarm:=(tRamp.Y+Loop.Config.Temp_Window_Alarm);
TT.Alarm_Config.Setpoints.Low_Low_Alarm:=(tRamp.Y-Loop.Config.Temp_Window_Alarm);
Loop.Live_Temp	:=tRamp.Y;
Temp_PID(In:=tRamp.Y-TT.EU,RST:=FALSE);



HW.PLC_CMD:= LIMIT(0, ((1+(Temp_PID.Y/100)) * Flow_PID.Y),100);
CW.PLC_CMD:= LIMIT(0, ((1-(Temp_PID.Y/100)) * Flow_PID.Y),100);



IF (FIT.Total> Loop.Target_Volume) THEN
	Loop.Status:=eQuick_Mix_Status.Batch_Complete;
END_IF
END_ACTION

ACTION Ramp_Up_active:
Flow_PID.KP:=Loop.Config.Flow_KP;
Flow_PID.TN:=Loop.Config.Flow_TN;
Flow_PID.TV:=Loop.Config.Flow_TV;
Flow_pid.LIM_L:=0;
Flow_PID.LIM_H:=100;

Temp_PID.KP:=Loop.Config.Temp_KP;
Temp_PID.TN:=Loop.Config.Temp_TN;
Temp_PID.TV:=Loop.Config.Temp_TV;
Temp_pid.LIM_L:=(-100);
Temp_PID.LIM_H:=100;





Loop.Status:=eQuick_Mix_Status.Start_Flow;
Loop.Active:=TRUE;
Ramp(x:=Loop.Target_Rate, Rst:=FALSE);
FIT.Rate.Alarm_Config.Setpoints.Alarm_Debounce	:=loop.Config.Alarm_Debounce;
FIT.Rate.Alarm_Config.Setpoints.Hi_Warn:=( Ramp.Y+ loop.Config.Flow_WIndow_Warn);
FIT.Rate.Alarm_Config.Setpoints.Low_Warn:=( Ramp.y- loop.Config.Flow_WIndow_Warn);
FIT.Rate.Alarm_Config.Setpoints.Hi_Hi_Alarm:=(Ramp.Y+Loop.Config.Flow_Window_Alarm);
FIT.Rate.Alarm_Config.Setpoints.Low_Low_Alarm:=(Ramp.Y-Loop.Config.Flow_Window_Alarm);
Flow_PID(In:=Ramp.Y-FIT.Rate.EU,RST:=NOT(Destination_OK));

tRamp(x:=Loop.Target_Temp, Rst:=FALSE);
TT.Alarm_Config.Setpoints.Hi_Warn:=( tRamp.Y+ loop.Config.Temp_WIndow_Warn);
TT.Alarm_Config.Setpoints.Low_Warn:=( tRamp.Y- loop.Config.Temp_WIndow_Warn);
TT.Alarm_Config.Setpoints.Hi_Hi_Alarm:=(tRamp.Y+Loop.Config.Temp_Window_Alarm);
TT.Alarm_Config.Setpoints.Low_Low_Alarm:=(tRamp.Y-Loop.Config.Temp_Window_Alarm);
Loop.Live_Temp	:=tRamp.Y;
Temp_PID(In:=tRamp.Y-TT.EU,RST:=NOT(Destination_OK));



Loop.Live_Rate:=Ramp.Y;


Ramp_Time:=(Ramp_UP.t);
Loop.ETA:=TO_INT((Loop.Target_Volume/Loop.Target_Rate)*60);
IF Ramp.Y = Ramp.X AND FIT.Rate.EU> Loop.Config.Min_Flow THEN
	Loop.Status:=eQuick_Mix_Status.Main_Rate;
END_IF;

//Loop.ETA:=0;

tHW:=((1+(Temp_PID.Y/100)) * Flow_PID.Y);
HW.PLC_CMD:= LIMIT(0, ((1+(Temp_PID.Y/100)) * Flow_PID.Y),100);
CW.PLC_CMD:= LIMIT(0, ((1-(Temp_PID.Y/100)) * Flow_PID.Y),100);


//HW.PLC_CMD:= Flow_PID.Y * (Temp_PID.y/100);
//CW.PLC_CMD:= Flow_PID.y * (1- (Temp_PID.y/100));
END_ACTION

ACTION Start_active:
IF Destination_OK THEN
	HW.PLC_CMD:=0;
	CW.PLC_CMD:=0;
END_IF;
END_ACTION

ACTION Start_entry:
HW.PLC_CMD:=0;
CW.PLC_CMD:=0;
Flow_PiD.PLC_Enable:=FALSE;
Temp_PID(RST:=TRUE);
Loop.ETA:=0;
Loop.Active:=FALSE;
Loop.Actual_Rate:=0;
END_ACTION

ACTION System_Test_active:
(*
Flow_PID.KP:=Loop.Config.Flow_KP;
Flow_PID.TN:=Loop.Config.Flow_TN;
Flow_PID.TV:=Loop.Config.Flow_TV;
Flow_pid.LIM_L:=0;
Flow_PID.LIM_H:=100;
*)
Temp_PID.KP:=Loop.Config.Temp_KP;
Temp_PID.TN:=Loop.Config.Temp_TN;
Temp_PID.TV:=Loop.Config.Temp_TV;
Temp_pid.LIM_L:=(-100);
Temp_PID.LIM_H:=100;



Loop.Status:=eQuick_Mix_Status.Fit_Reset;
Loop.Active:=TRUE;
IF NOT(HW.Ready) THEN
	Loop.Status:=eQuick_Mix_Status.HW_Not_Ready;
END_IF;


IF NOT(CW.Ready) THEN
	Loop.Status:=eQuick_Mix_Status.CW_Not_Ready;
END_IF;


IF NOT(TT.Ready) THEN
	Loop.Status:=eQuick_Mix_Status.TT_Not_Ready;
END_IF;

IF FIT.Rate.EU > 1 THEN
	Loop.Status:=eQuick_Mix_Status.Flow_Not_Ready;
END_IF;

IF NOT(Destination_Ok) THEN
	Loop.Status:= eQuick_Mix_Status.Destination_Not_Ready;
END_IF;
END_ACTION

ACTION System_Text_entry:
Loop.ETA:=TO_INT((Loop.Target_Volume/Loop.Target_Rate)*60);
END_ACTION

END_FUNCTION_BLOCK

// Level_2_Controls/Rate_Batch
FUNCTION_BLOCK Rate_Batch
VAR_INPUT
	Config: REFERENCE TO cBatch;
	Rate_PID:	REFERENCE TO PID_Control;
	Volume_PID:	REFERENCE TO PID_Control;
	FIT:	REFERENCE TO Burkert.cFIT;
	
	CV_OK:BOOL;
END_VAR
VAR_OUTPUT
	CV:REAL;
END_VAR
VAR
	Local_Mode:Burkert.eHOA_Modes;
	Local_Task:eBatch_Task;
	Local_Status:eBatch_Status;
	
	Start_Rate:REAL;
	Main_Rate:REAL;
	End_Rate:REAL;
	
	
	Batch_Duration_S:UINT;
	clk_250:Burkert_OSCAT_BASIC.CLK_PRG;
	Batch_Clock_S:REAL;
	
END_VAR

CASE Config.Mode.eMode OF
	Burkert.eHOA_Modes.Off:		Mode_OFF();
	Burkert.eHOA_Modes.Manual:	Mode_Manual();
	Burkert.eHOA_Modes.Auto:	Mode_Auto();	
END_CASE


CASE Config.Task OF
	eBatch_task.OFF	: 	Task_OFf();
	eBatch_task.Pause :	Task_Pause();
	eBatch_Task.Resume: Task_Resume();
	eBatch_task.Run:	Task_Run();
END_CASE

END_FUNCTION_BLOCK

// Level_2_Controls/SW_CTRL_ACV
FUNCTION_BLOCK SW_CTRL_ACV 
VAR_INPUT
	SW: REFERENCE TO cBatch_Transfer;
	FIT:REFERENCE TO Burkert.cFIT;
	ACV:REFERENCE TO Burkert.cACV;
	Pump_Ready:BOOL;
	Interlock:BOOL;
END_VAR
VAR
	PID: BURKERT_OSCAT_BASIC.FT_PIDW;
END_VAR

IF (
		(
		(SW.Auto_Batch = FALSE AND SW.Mode.eMode=eBatch_Transfer_Mode.Auto) OR
		(SW.Mode.eMode=eBatch_Transfer_Mode.Disabled) 
		)
			AND SW.Status<> Transfer_Status.IDLE 
			
	) THEN
	SW.Status:=Transfer_Status.IDLE;
	
END_IF;

IF (FIT.Rate.EU>1 AND NOT(ACV.Status.eStatus=Burkert.eBCV_Status.A_Open) AND NOT(Interlock) AND NOT(SW.Status=Transfer_Status.Complete) )THEN
	SW.Status:=Transfer_Status.Flow_Meter_Active;
	SW.Ready:=FALSE;
	SW.Active:=FALSE;
END_IF;

IF NOT(Pump_Ready) THEN
	SW.Status:=Transfer_Status.Pump_Not_Ready;
	SW.Ready:=FALSE;
	SW.Active:=FALSE;
END_IF


IF NOT(ACV.Ready) THEN
	SW.Status:=Transfer_Status.BCV_Not_Ready;
	SW.Ready:=FALSE;
	SW.Active:=FALSE;
END_IF;

IF (ACV.Status.eStatus=Burkert.eBCV_Status.Interlocked OR ACV.Status.eStatus=Burkert.eBCV_Status.LOCKED_OUT ) THEN
	SW.Status:=Transfer_Status.LOCKED_OUT;
	SW.Ready:=FALSE;
	SW.Active:=FALSE;
END_IF;


IF Sw.Status=Transfer_Status.IDLE AND Interlock THEN
	SW.Status:=Transfer_Status.LOCKED_OUT;
END_IF

CASE SW.Status OF
	
	Transfer_Status.IDLE:
		SW.Ready:=TRUE;
		//SW.BCV:=FALSE;
		
		SW.Remaining_Time_S:=0;
		SW.Current_Rate:=0;
		SW.Current_Volume:=0;
		SW.Remaining_Volume:=0;
		SW.Active:=FALSE;
		
		IF (
			(SW.Auto_Batch AND SW.Mode.eMode=eBatch_Transfer_Mode.Auto) OR
			( SW.Mode.eMode=eBatch_Transfer_Mode.Batch)
			)THEN
			SW.Status:=Transfer_Status.FIT_Reset;
		END_IF;
		
		
	Transfer_Status.FIT_Reset:
		SW.Active:=TRUE;
		//SW.BCV:=FALSE;
		SW.Remaining_Time_S:=0;
		FIT.PLC_Reset:=(FIT.Total>1);
		IF FIT.Total<1 THEN
			SW.Status:=Transfer_Status.Open_Valve;
		END_IF;
		
	Transfer_Status.Open_Valve:
	//SW.BCV:=TRUE;
	//IF SW.ACV AND ACV.Valve_Actual>10 THEN
			SW.Status:=Transfer_Status.Flow_Active;	
		//END_IF;
		
	
		
	Transfer_Status.Flow_Active:
		//SW.BCV:=TRUE;
		SW.Remaining_Time_S:=TO_UDINT(SW.Remaining_Volume/(FIT.Rate.EU/60));
		SW.Current_Rate:=FIT.Rate.EU;
		SW.Current_Volume:=FIT.Total;
		SW.Remaining_Volume:=(SW.Volume-FIT.Total);
		
		
		IF (
			(FIT.Rate.EU > (SW.Rate*0.25)) OR
			(FIT.Total> (SW.Volume*0.80))
		) THEN
			SW.Status:=Transfer_Status.Running;
		END_IF;
	Transfer_Status.Running:	
			//SW.BCV:=TRUE;
			SW.Remaining_Time_S:=TO_UDINT(SW.Remaining_Volume/(FIT.Rate.EU/60));
			SW.Current_Rate:=FIT.Rate.EU;
			SW.Current_Volume:=FIT.Total;	
			SW.Remaining_Volume:=(SW.Volume-FIT.Total);
			IF (FIT.Total> SW.Volume)
			THEN
				SW.Status:=Transfer_Status.Complete;
			END_IF;
	Transfer_Status.Complete:
		//SW.BCV:=FALSE;
		SW.Remaining_Time_S:=0;
		SW.Current_Rate:=0;
		SW.Current_Volume:=0;
		SW.Remaining_Volume:=0;
		SW.Active:=FALSE;
		
	Transfer_Status.LOCKED_OUT:
		SW.Ready:=FALSE;
		SW.Active:=FALSE;
		SW.Remaining_Time_S:=0;
		SW.Current_Rate:=0;
		SW.Current_Volume:=0;
		SW.Remaining_Volume:=0;
		
		
	Transfer_Status.Destination_Not_Ready:
		//SW.Active:=FALSE;
		IF ACV.Ready THEN
			SW.Status:=Transfer_Status.Flow_Active;		
		END_IF;
		IF 	(
				NOT(SW.Mode.eMode=eBatch_Transfer_mode.Auto AND SW.Auto_Batch = TRUE) AND
				NOT(SW.Mode.eMode=eBatch_Transfer_mode.Batch) AND
				SW.BCV=TRUE
			)THEN
			SW.BCV:=FALSE;
		END_IF;
	Transfer_Status.Flow_Meter_Active:
		IF FIT.Rate.EU<0.5 THEN
			SW.Status:=Transfer_Status.IDLE;
		END_IF;
END_CASE;



PID(
	IN:= (SW.Rate-FIT.Rate.EU), 
	KP:= SW.Config.KP, 
	TN:= SW.Config.TN, 
	TV:= SW.Config.TV, 
	LIM_L:= 0, 
	LIM_H:= 100-(SW.Config.FF*SW.Rate), 
	RST:= NOT(SW.Active) OR NOT(ACV.Ready) , 
	Y=> , 
	LIM=> );
	
IF NOT(SW.Active) THEN
	SW.ACV:=0;
	ACV.PLC_CMD:=0;
	//SW.BCV:=FALSE;
ELSE
	SW.ACV:=PID.Y+(SW.Config.FF*SW.Rate);
	ACV.PLC_CMD:=SW.ACV;
END_IF;

END_FUNCTION_BLOCK

// Level_2_Controls/SW_CTRL
FUNCTION_BLOCK SW_CTRL 
VAR_INPUT
	SW: REFERENCE TO cBatch_Transfer;
	FIT:REFERENCE TO Burkert.cFIT;
	BCV:REFERENCE TO Burkert.cBCV;
	Pump_Ready:BOOL;
	Interlock:BOOL;
END_VAR
VAR
	PID: BURKERT_OSCAT_BASIC.FT_PIDW;
END_VAR

IF (
		(
		(SW.Auto_Batch = FALSE AND SW.Mode.eMode=eBatch_Transfer_Mode.Auto) OR
		(SW.Mode.eMode=eBatch_Transfer_Mode.Disabled) 
		)
			AND SW.Status<> Transfer_Status.IDLE 
			
	) THEN
	SW.Status:=Transfer_Status.IDLE;
	
END_IF;

IF (FIT.Rate.EU>1 AND NOT(BCV.Status.eStatus=Burkert.eBCV_Status.A_Open) AND NOT(Interlock) AND NOT(SW.Status=Transfer_Status.Complete) )THEN
	SW.Status:=Transfer_Status.Flow_Meter_Active;
	SW.Ready:=FALSE;
	SW.Active:=FALSE;
END_IF;

IF NOT(Pump_Ready) THEN
	SW.Status:=Transfer_Status.Pump_Not_Ready;
	SW.Ready:=FALSE;
	SW.Active:=FALSE;
END_IF


IF NOT(BCV.Ready) THEN
	SW.Status:=Transfer_Status.BCV_Not_Ready;
	SW.Ready:=FALSE;
	SW.Active:=FALSE;
END_IF;

IF (BCV.Status.eStatus=Burkert.eBCV_Status.Interlocked OR BCV.Status.eStatus=Burkert.eBCV_Status.LOCKED_OUT ) THEN
	SW.Status:=Transfer_Status.LOCKED_OUT;
	SW.Ready:=FALSE;
	SW.Active:=FALSE;
END_IF;


IF Sw.Status=Transfer_Status.IDLE AND Interlock THEN
	SW.Status:=Transfer_Status.LOCKED_OUT;
END_IF

CASE SW.Status OF
	
	Transfer_Status.IDLE:
		SW.Ready:=TRUE;
		SW.BCV:=FALSE;
		
		SW.Remaining_Time_S:=0;
		SW.Current_Rate:=0;
		SW.Current_Volume:=0;
		SW.Remaining_Volume:=0;
		SW.Active:=FALSE;
		
		IF (
			(SW.Auto_Batch AND SW.Mode.eMode=eBatch_Transfer_Mode.Auto) OR
			( SW.Mode.eMode=eBatch_Transfer_Mode.Batch)
			)THEN
			SW.Status:=Transfer_Status.FIT_Reset;
		END_IF;
		
		
	Transfer_Status.FIT_Reset:
		SW.Active:=TRUE;
		SW.BCV:=FALSE;
		SW.Remaining_Time_S:=0;
		FIT.PLC_Reset:=(FIT.Total>1);
		IF FIT.Total<1 THEN
			SW.Status:=Transfer_Status.Open_Valve;
		END_IF;
		
	Transfer_Status.Open_Valve:
	SW.BCV:=TRUE;
	IF SW.BCV AND BCV.Status.eStatus=Burkert.eBCV_Status.A_Open THEN
			SW.Status:=Transfer_Status.Flow_Active;	
		END_IF;
		
	
		
	Transfer_Status.Flow_Active:
		SW.BCV:=TRUE;
		SW.Remaining_Time_S:=TO_UDINT(SW.Remaining_Volume/(FIT.Rate.EU/60));
		SW.Current_Rate:=FIT.Rate.EU;
		SW.Current_Volume:=FIT.Total;
		SW.Remaining_Volume:=(SW.Volume-FIT.Total);
		
		
		IF (
			(FIT.Rate.EU > (SW.Rate*0.25)) OR
			(FIT.Total> (SW.Volume*0.80))
		) THEN
			SW.Status:=Transfer_Status.Running;
		END_IF;
	Transfer_Status.Running:	
			SW.BCV:=TRUE;
			SW.Remaining_Time_S:=TO_UDINT(SW.Remaining_Volume/(FIT.Rate.EU/60));
			SW.Current_Rate:=FIT.Rate.EU;
			SW.Current_Volume:=FIT.Total;	
			SW.Remaining_Volume:=(SW.Volume-FIT.Total);
			IF (FIT.Total> SW.Volume)
			THEN
				SW.Status:=Transfer_Status.Complete;
			END_IF;
	Transfer_Status.Complete:
		SW.BCV:=FALSE;
		SW.Remaining_Time_S:=0;
		SW.Current_Rate:=0;
		SW.Current_Volume:=0;
		SW.Remaining_Volume:=0;
		SW.Active:=FALSE;
		
	Transfer_Status.LOCKED_OUT:
		SW.Ready:=FALSE;
		SW.Active:=FALSE;
		SW.Remaining_Time_S:=0;
		SW.Current_Rate:=0;
		SW.Current_Volume:=0;
		SW.Remaining_Volume:=0;
		
		
	Transfer_Status.Destination_Not_Ready:
		SW.Active:=FALSE;
		IF SW.BCV AND BCV.Status.eStatus=Burkert.eBCV_Status.A_Open THEN
			SW.Status:=Transfer_Status.Flow_Active;		
		END_IF;
		IF 	(
				NOT(SW.Mode.eMode=eBatch_Transfer_mode.Auto AND SW.Auto_Batch = TRUE) AND
				NOT(SW.Mode.eMode=eBatch_Transfer_mode.Batch) AND
				SW.BCV=TRUE
			)THEN
			SW.BCV:=FALSE;
		END_IF;
	Transfer_Status.Flow_Meter_Active:
		IF FIT.Rate.EU<0.5 THEN
			SW.Status:=Transfer_Status.IDLE;
		END_IF;
END_CASE;



PID(
	IN:= (SW.Rate-FIT.Rate.EU), 
	KP:= SW.Config.KP, 
	TN:= SW.Config.TN, 
	TV:= SW.Config.TV, 
	LIM_L:= 0, 
	LIM_H:= 100-(SW.Config.FF*SW.Rate), 
	RST:= NOT(SW.Active) OR NOT(BCV.Status.eStatus=Burkert.eBCV_Status.A_Open) , 
	Y=> , 
	LIM=> );
	
IF NOT(SW.Active) THEN
	SW.ACV:=0;
	SW.BCV:=FALSE;
ELSE
	SW.ACV:=PID.Y+(SW.Config.FF*SW.Rate);

END_IF;

END_FUNCTION_BLOCK

// Level_2_Controls/Tempered_Line_4_Valve
FUNCTION_BLOCK Tempered_Line_4_Valve
VAR_INPUT
	Config_DATA:REFERENCE TO 		cTempered_Line_Data;
	
	HW_Supply_TT:REFERENCE TO 		Burkert.cSensor;
	CW_Supply_TT:REFERENCE TO 		Burkert.cSensor;
	
	CW_Inlet_PT:REFERENCE TO 		Burkert.cSensor;
	CW_Outlet_PT:REFERENCE TO 		Burkert.cSensor;
	HW_Inlet_PT:REFERENCE TO 			Burkert.cSensor;
	HW_Outlet_PT:REFERENCE TO 		Burkert.cSensor;
	Combined_Temp:REFERENCE TO 		Burkert.cSensor;
	
	HW_FIT:REFERENCE TO 			Burkert.cFIT;
	CW_FIT:REFERENCE TO 		Burkert.cFIT;

	HW_PID		:REFERENCE TO PID_DUT;
	CW_PID		:REFERENCE TO PID_DUT;
	Temperature_PID		:REFERENCE TO PID_DUT;
	
	CW1_ACV		:REFERENCE TO Burkert.cACV;
	CW2_ACV		:REFERENCE TO Burkert.cACV;
	HW1_ACV		:REFERENCE TO Burkert.cACV;
	HW2_ACV		:REFERENCE TO Burkert.cACV;
	
	KV_Curve	:REFERENCE TO ARRAY[0..100] OF REAL;
	CV_2_KV		:REFERENCE TO ARRAY[0..100] OF REAL;
	
	Temp_Flow_CV	:REFERENCE TO cTempered_C;
	
	Flow_Units:eUnits;
	Temperature_Units:eUnits;
	Run_mode:BYTE;
	
	
	HW_CV_Mode_3:INT;
	CW_CV_Mode_3:INT;
	
	Min_Flow:REAL:=0.5;
	
END_VAR
VAR_OUTPUT
END_VAR
VAR
	Local_Mode:eTempered_modes;
	Local_Task:eTempered_Task;
	Local_Status:eTempered_Status;
	On_Target:BOOL;
	Task_Ton:Ton;
	Prepare_TON:TON;
	
	
	Temp_Index:INT;
	Flow_Index:INT;
	
	CW_KV_Index:INT;
	HW_KV_Index:INT;
	
	CW_Target_KV_Index:INT;
	HW_Target_KV_Index:INT;
	
	Calibration_Temp:Burkert.cAlarm_Window;
	
	
	KV_Index_Scalar:INT:=20;
	
	HW_CV_Ramp:RAMP_REAL;
	CW_CV_Ramp:RAMP_REAL;
	
	TOF_0: TOF;
	Valid:BOOL;
END_VAR
VAR // added by the converter: edge detectors and wires of the graphical bodies
    _w1, _w2 : ANY;
END_VAR

Valid:=(
	__ISVALIDREF(CW_FIT) AND
	__ISVALIDREF(HW_FIT)
	);
	
IF Valid THEN	
	AUX();
	Alarms();
	Math();
	PID_CTRL();
	ACV_CTRL();
END_IF;


Task_Ton();

ACTION Alarms:

(*
HW_FIT.Rate.Alarm_Config.Setpoints.Hi_Hi_Alarm	:=Config_Data.HW_Target_Flow+Config.Min_Flow.Alarm_Window;
HW_FIT.Rate.Alarm_Config.Setpoints.Hi_Warn		:=Config_Data.HW_Target_Flow+Config.Min_Flow.Warn_Window;
HW_FIT.Rate.Alarm_Config.Setpoints.Low_Warn		:=Config_Data.HW_Target_Flow-Config.Min_Flow.Warn_Window;
HW_FIT.Rate.Alarm_Config.Setpoints.Low_Low_Alarm		:=Config_Data.HW_Target_Flow-Config.Min_Flow.Alarm_Window;
HW_FIT.Rate.Alarm_Config.Debounce			:=Config.Min_Flow.Alarm_Delay;
HW_Fit.Rate.Alarm_Config.Silence:=HW_PID.CV<5;

CW_FIT.Rate.Alarm_Config.Setpoints.Hi_Hi_Alarm	:=Config_Data.CW_Target_Flow+Config.Min_Flow.Alarm_Window;
CW_FIT.Rate.Alarm_Config.Setpoints.Hi_Warn		:=Config_Data.CW_Target_Flow+Config.Min_Flow.Warn_Window;
CW_FIT.Rate.Alarm_Config.Setpoints.Low_Warn		:=Config_Data.CW_Target_Flow-Config.Min_Flow.Warn_Window;
CW_FIT.Rate.Alarm_Config.Setpoints.Low_Low_Alarm		:=Config_Data.CW_Target_Flow-Config.Min_Flow.Alarm_Window;
CW_FIT.Rate.Alarm_Config.Debounce			:=Config_Min_Flow.Alarm_Delay;
CW_Fit.Rate.Alarm_Config.Silence:=CW_PID.CV<5;
*)

//Pressure.Burkert.cAlarm_Config:=Alarm_Window_Convert(Config.Target_Pressure);
//Drain_FIT.Rate.Alarm_Config:=Alarm_Window_Convert(Config.Min_Flow);
//Combined_Temp.Burkert.cAlarm_Config:=Alarm_Window_Convert(Config.Target_Temp);




CASE Local_Task OF
	eTempered_Task.Calibrate:
		HW_Fit.Rate.Alarm_Config.Silence:=Config_Data.Mode=eTempered_modes.CW_Only;
		CW_Fit.Rate.Alarm_Config.Silence:=Config_Data.Mode=eTempered_modes.HW_Only;
		Combined_temp.Alarm_Config.Silence:=FALSE;;
	eTempered_Task.Drain:
		HW_Fit.Rate.Alarm_Config.Silence:=TRUE;
		CW_Fit.Rate.Alarm_Config.Silence:=TRUE;
		Combined_temp.Alarm_Config.Silence:=TRUE;
	eTempered_Task.OFF:
		HW_Fit.Rate.Alarm_Config.Silence:=TRUE;
		CW_Fit.Rate.Alarm_Config.Silence:=TRUE;
		Combined_temp.Alarm_Config.Silence:=TRUE;
	eTempered_Task.Prime:
		HW_Fit.Rate.Alarm_Config.Silence:=Config_Data.Mode=eTempered_modes.CW_Only ;
		CW_Fit.Rate.Alarm_Config.Silence:=Config_Data.Mode=eTempered_modes.HW_Only;
		Combined_temp.Alarm_Config.Silence:=FALSE;
	eTempered_Task.Run:
		HW_Fit.Rate.Alarm_Config.Silence:=Config_Data.Mode=eTempered_modes.CW_Only;
		CW_Fit.Rate.Alarm_Config.Silence:=Config_Data.Mode=eTempered_modes.HW_Only;
		Combined_temp.Alarm_Config.Silence:=FALSE;
END_CASE;
END_ACTION

ACTION AUX:
HW_PID.Actual:=HW_FIT.Rate.EU;
CW_PID.Actual:=CW_FIT.Rate.EU;
Temperature_PID.Actual:=Combined_temp.EU;

HW_PID.PLC_Target:=Config_Data.HW_Target_Flow;
CW_PID.PLC_Target:=Config_Data.CW_Target_Flow;





Config_Data.CW_Flow_OK:=			CW_FIT.Rate.Alarm_Config.Within_Norms;//		(CW_FIT.Rate.Status.eStatus	=		Burkert.eSensor_Status.OK); //AND ABS(CW_PID.Err)<Config.Min_Flow.Warn_Window;
COnfig_Data.HW_Flow_OK:=			HW_FIT.Rate.Alarm_Config.Within_Norms;//		(HW_FIT.Rate.Status.eStatus	=		Burkert.eSensor_Status.OK); //AND ABS(HW_PID.Err)<Config.Min_Flow.Warn_Window;;
Config_Data.Temperature_OK:=		Combined_temp.Alarm_Config.Within_Norms;	//	Combined_temp.Status.eStatus=		Burkert.eSensor_Status.OK;


Config_Data.StrStatus:= Burkert_OSCAT_BASIC.REPLACE_ALL(str:=TO_STRING(Config_Data.Status.eStatus) , src:='_' , rep:=' ' );


//Burkert.Burkert.eSensor_Status.OK


Config_Data.CW_CV:=CW_PID.CV;
Config_Data.HW_CV:=HW_PID.CV;
Config_Data.Flow_Rate:=(HW_FIT.Rate.EU+CW_FIT.Rate.EU);
Config_Data.Total_Volume:=(CW_FIT.Total+HW_FIT.Total);
Config_Data.Temperature:=Combined_Temp.EU;
(*
IF CW_PID.CV>0 THEN
	Config_Data.CW_FF:=	(CW_PID.PLC_Target/CW_PID.CV);
END_IF;
IF HW_PID.CV>0 THEN	
	Config_Data.HW_FF:=	(HW_PID.PLC_Target/HW_PID.CV);
END_IF;

*)



//Temperature_PID.PLC_Target:=Config_Data.Target_Temperature;
//Temperature_PID.FF:=1;
Temperature_PID.CV_Min:=(CW_Supply_TT.EU*1.0);
Temperature_PID.CV_Max:=(HW_Supply_TT.EU*1);


Config_Data.HW_DP:=HW_Inlet_PT.EU-HW_Outlet_PT.EU;
Config_Data.CW_DP:=CW_Inlet_PT.EU-CW_Outlet_PT.EU;


Config_Data.CW_Target_KV:=KV_Calculator(FR:=Unit_Convert(eFrom:=Flow_Units,eTo:=eUnits.lpm,Source:= Config_Data.CW_Target_Flow) ,DeltaP:=Config_Data.CW_DP,SG:=1);
Config_Data.HW_Target_KV:=KV_Calculator(FR:=Unit_Convert(eFrom:=Flow_Units,eTo:=eUnits.lpm,Source:= Config_Data.HW_Target_Flow) ,DeltaP:=Config_Data.HW_DP,SG:=1);

Config_Data.CW_KV:=KV_Calculator(FR:=Unit_Convert(eFrom:=Flow_Units,eTo:=eUnits.lpm,Source:= CW_FIT.Rate.EU) ,DeltaP:=Config_Data.CW_DP,SG:=1);
Config_Data.HW_KV:=KV_Calculator(FR:=Unit_Convert(eFrom:=Flow_Units,eTo:=eUnits.lpm,Source:= HW_FIT.Rate.EU) ,DeltaP:=Config_Data.HW_DP,SG:=1);

HW_KV_Index:=LIMIT(0,TO_INT(Config_Data.HW_KV*KV_Index_Scalar),100);
CW_KV_Index:=LIMIT(0,TO_INT(Config_Data.CW_KV*KV_Index_Scalar),100);

HW_Target_KV_Index:=LIMIT(0,TO_INT(Config_Data.HW_Target_KV*KV_Index_Scalar),100);
CW_Target_KV_Index:=LIMIT(0,TO_INT(Config_Data.CW_Target_KV*KV_Index_Scalar),100);


HW_CV_Ramp(ASCEND:=1,Descend:=1,TimeBase:=T#1S);
CW_CV_Ramp(ASCEND:=1,Descend:=1,TimeBase:=T#1S);
END_ACTION

ACTION Math:
IF Config_Data.Base_Flow>0 AND HW_Supply_TT.EU>CW_Supply_TT.eu  THEN
	CASE Config_Data.Mode OF
		eTempered_modes.Mix:
			Tempered_Flow_Calculator(
				CT:=CW_Supply_TT.EU,
				HT:=HW_Supply_TT.EU,
				Required_Flow:=Config_Data.Base_Flow,
				Required_Temperature:=Config_Data.Target_Temperature,
				Hot_Flow =>Config_Data.HW_Target_Flow,
				Cold_Flow =>Config_Data.CW_Target_Flow);
		eTempered_modes.HW_Only:
			Config_Data.HW_Target_Flow:=Config_Data.Base_Flow;
			Config_Data.CW_Target_Flow:=0;
		eTempered_modes.CW_Only:
			Config_Data.HW_Target_Flow:=0;
			Config_Data.CW_Target_Flow:=Config_Data.Base_Flow;
	END_CASE
ELSE
	Config_Data.CW_Target_Flow:=Config_Data.Base_Flow/2;
	Config_Data.HW_Target_Flow:=Config_Data.Base_Flow/2;
END_IF;
END_ACTION

ACTION PID_CTRL:
_w1 := (Config_data.Status.eStatus=eTempered_Status.Prepare_Standby) OR (Config_data.Status.eStatus=eTempered_Status.Prepare_Active) OR (Config_Data.Status.eStatus=eTempered_Status.Prepare_Complete) OR (Config_data.Status.eStatus=eTempered_Status.Starting) OR (Config_Data.Status.eStatus=eTempered_Status.Ready);
_w2 := _w1 OR (Config_Data.Status.eStatus=eTempered_Status.Prime_Start) OR (Config_Data.Status.eStatus=eTempered_Status.Prime_Active) OR (Config_Data.Status.eStatus=eTempered_Status.Prime_Complete);
HW_PID.PLC_Enable := _w2;
CW_PID.PLC_Enable := _w2;
TOF_0(IN := (HW_Supply_TT.Status.eStatus=Burkert.eSensor_Status.OK) AND (CW_Supply_TT.Status.eStatus=Burkert.eSensor_Status.OK) AND (HW_FIT.Rate.EU>0.2) AND (CW_FIT.Rate.EU>0.2) AND _w1, PT := T#2s); // TOF
Temperature_PID.PLC_Enable := TOF_0.Q;
END_ACTION

METHOD Task_Calibrate : BOOL
VAR_INPUT
	Rate:Burkert.cAlarm_Window;
	Temperature:Burkert.cAlarm_Window;
END_VAR

VAR

END_VAR
IF Local_Task<>eTempered_Task.Calibrate THEN
	Local_Task:=eTempered_Task.Calibrate;
	Local_Status:=eTempered_Status.Prepare_Standby;
	HW_PID.FF:=0;
	CW_PID.FF:=0;
	ON_Target:=FALSE;
	Config_Data.Max_Flow:=0;
	Calibration_Temp:=Temperature;
	
	Calibration_temp.Alarm_Window:=Temperature.Alarm_Window/2;
	Calibration_Temp.Warn_Window:=Temperature.Warn_Window/2;
	Burkert.Alarm_Window_Convert(	Window:=Calibration_Temp,	Config:=Combined_Temp.Alarm_Config);
	Task_Ton.PT:=T#5S;
	
END_IF;

AUX();
Alarms();
Math();
PID_CTRL();
ACV_CTRL();

Task_Ton();

CASE Config_Data.Mode OF
	eTempered_modes.Mix:		Temperature_PID.PLC_Target:=Temperature.Target;
	eTempered_modes.CW_Only:	Temperature_PID.PLC_Target:=CW_Supply_TT.EU;
	eTempered_modes.HW_Only:	Temperature_PID.PLC_Target:=HW_Supply_TT.EU;
END_CASE;

Config_Data.Base_Flow:=Rate.Target;
IF Temperature_PID.PLC_Enable THEN
	Config_Data.Target_Temperature:= Temperature_PID.CV;
ELSE
	Config_Data.Target_Temperature:= Temperature_PID.PLC_Target;
END_IF;

Config_Data.Target_Volume:=9999;

HW_FIT.Rate.Alarm_Config.Setpoints.Hi_Hi_Alarm	:=Config_Data.HW_Target_Flow+Rate.Alarm_Window;
HW_FIT.Rate.Alarm_Config.Setpoints.Hi_Warn		:=Config_Data.HW_Target_Flow+Rate.Warn_Window;
HW_FIT.Rate.Alarm_Config.Setpoints.Low_Warn		:=Config_Data.HW_Target_Flow-Rate.Warn_Window;
HW_FIT.Rate.Alarm_Config.Setpoints.Low_Low_Alarm		:=Config_Data.HW_Target_Flow-Rate.Alarm_Window;
HW_FIT.Rate.Alarm_Config.Setpoints.Alarm_Debounce			:=Rate.Alarm_Delay;
HW_FIT.Rate.Alarm_Config.Setpoints.Warn_Debounce		:=(Rate.Alarm_Delay/2);
HW_Fit.Rate.Alarm_Config.Silence:=NOT(HW_PID.PLC_Enable);

CW_FIT.Rate.Alarm_Config.Setpoints.Hi_Hi_Alarm	:=Config_Data.CW_Target_Flow+Rate.Alarm_Window;
CW_FIT.Rate.Alarm_Config.Setpoints.Hi_Warn		:=Config_Data.CW_Target_Flow+Rate.Warn_Window;
CW_FIT.Rate.Alarm_Config.Setpoints.Low_Warn		:=Config_Data.CW_Target_Flow-Rate.Warn_Window;
CW_FIT.Rate.Alarm_Config.Setpoints.Low_Low_Alarm		:=Config_Data.CW_Target_Flow-Rate.Alarm_Window;
CW_FIT.Rate.Alarm_Config.Setpoints.Alarm_Debounce			:=Rate.Alarm_Delay;
CW_FIT.Rate.Alarm_Config.Setpoints.Warn_Debounce			:=Rate.Alarm_Delay/2;
CW_Fit.Rate.Alarm_Config.Silence:=NOT(CW_PID.PLC_Enable);

Combined_temp.Alarm_Config.Setpoints.Alarm_Debounce:=0;
Combined_temp.Alarm_Config.Setpoints.Warn_Debounce:=0;



Config_data.Status.eStatus:=Status_Test(Local_Status);


Performance_Check();

Temp_index:=LIMIT(20,TO_INT(Unit_Convert(eFrom:=Temperature_Units,eTO:=eUnits.C,Source:= Temperature.Target)),60);
Flow_index:=LIMIT(10,TO_INT(Unit_Convert(eFrom:=Flow_units,eTo:=Eunits.lpm,Source:= CW_FIT.Rate.EU+HW_FIT.Rate.EU)),60);

CASE Config_Data.Status.eStatus OF

	eTempered_Status.Prepare_Standby:
		Config_Data.Base_Flow:=Rate.Target;
		
		ON_Target:=FALSE;
		IF Config_Data.Flow_Rate>(Rate.Target*0.5) THEN
			Local_Status:=eTempered_Status.Prepare_Active;
		END_IF;
	eTempered_Status.Prepare_Active:
		IF Prepare_TON.Q THEN
			Local_Status:=eTempered_Status.Prepare_Complete;
		END_IF;
	eTempered_status.Prepare_Complete:
		Task_Calibrate:=On_Target;
END_CASE;
Prepare_TON(PT:=T#10S,IN:=(Config_data.Temperature_OK AND Config_Data.HW_Flow_OK AND Config_data.CW_Flow_OK));

IF CW1_ACV.Valve_Actual>95 AND  CW2_ACV.Valve_Actual>95 AND  HW1_ACV.Valve_Actual>95 AND  HW2_ACV.Valve_Actual>95 AND On_Target=FALSE  THEN

	Local_Status:=eTempered_Status.Prepare_Complete;
END_IF;
IF Config_Data.Flow_Rate>Config_Data.Max_Flow THEN
		Config_Data.Max_Flow:=Config_Data.Flow_Rate;
END_IF

	Store_Calibration();
END_METHOD

METHOD Task_Prime : BOOL
VAR_INPUT
	Rate:Burkert.cAlarm_Window;
	Temperature:Burkert.cAlarm_Window;
	Volume:REAL;
END_VAR


VAR
	Temp_C:INT;
	Flow_LPM:INT;
END_VAR
IF Local_Task<>eTempered_Task.Prime THEN
	Local_Task:=eTempered_Task.Prime;
	Local_Status:=eTempered_Status.Prime_Start;
	ON_Target:=FALSE;
	CW_PID.FF:=0.0;
	HW_PID.FF:=0.0;
	Task_Ton.PT:=T#120S;
	Task_Ton.IN:=FALSE;
END_IF;

AUX();
Alarms();
Math();
PID_CTRL();
ACV_CTRL();
Task_Ton();


CASE Config_Data.Mode OF
	eTempered_modes.Mix:		Temperature_PID.PLC_Target:=Temperature.Target;
	eTempered_modes.CW_Only:	Temperature_PID.PLC_Target:=CW_Supply_TT.EU;
	eTempered_modes.HW_Only:	Temperature_PID.PLC_Target:=HW_Supply_TT.EU;
END_CASE;

HW_FIT.Rate.Alarm_Config.Setpoints.Hi_Hi_Alarm			:=Config_Data.HW_Target_Flow+Rate.Alarm_Window;
HW_FIT.Rate.Alarm_Config.Setpoints.Hi_Warn				:=Config_Data.HW_Target_Flow+Rate.Warn_Window;
HW_FIT.Rate.Alarm_Config.Setpoints.Low_Warn				:=Config_Data.HW_Target_Flow-Rate.Warn_Window;
HW_FIT.Rate.Alarm_Config.Setpoints.Low_Low_Alarm			:=Config_Data.HW_Target_Flow-Rate.Alarm_Window;
HW_FIT.Rate.Alarm_Config.Setpoints.Alarm_Debounce			:=Rate.Alarm_Delay;
HW_FIT.Rate.Alarm_Config.Setpoints.Warn_Debounce			:=Rate.Alarm_Delay;
HW_Fit.Rate.Alarm_Config.Silence:=HW_PID.CV<2;

CW_FIT.Rate.Alarm_Config.Setpoints.Hi_Hi_Alarm			:=Config_Data.CW_Target_Flow+Rate.Alarm_Window;
CW_FIT.Rate.Alarm_Config.Setpoints.Hi_Warn				:=Config_Data.CW_Target_Flow+Rate.Warn_Window;
CW_FIT.Rate.Alarm_Config.Setpoints.Low_Warn				:=Config_Data.CW_Target_Flow-Rate.Warn_Window;
CW_FIT.Rate.Alarm_Config.Setpoints.Low_Low_Alarm			:=Config_Data.CW_Target_Flow-Rate.Alarm_Window;
CW_FIT.Rate.Alarm_Config.Setpoints.Alarm_Debounce			:=Rate.Alarm_Delay;
CW_FIT.Rate.Alarm_Config.Setpoints.Warn_Debounce			:=Rate.Alarm_Delay;
CW_Fit.Rate.Alarm_Config.Silence:=CW_PID.CV<2;

Burkert.Alarm_Window_Convert(Window:=Temperature,Config:=Combined_Temp.Alarm_Config);




Config_Data.Status.eStatus:=Status_Test(Local_Status);

Config_Data.Base_Flow:=Rate.Target;
Config_Data.Target_Temperature:= Temperature.Target;

CW_CV_Mode_3:=FindClosestIndexSorted(ArrayIn:=CV_2_KV,TargetValue:=Config_Data.CW_Target_KV);
HW_CV_Mode_3:=FindClosestIndexSorted(ArrayIn:=CV_2_KV,TargetValue:=Config_Data.HW_Target_KV);


//Task_Ton.IN:=Config_Data.HW_Flow_OK AND Config_Data.CW_Flow_OK;
CASE Run_mode OF
	
	0:
		CW_PID.FF:=0.0;
		HW_PID.FF:=0.0;
		Config_Data.HW_FF:=0;
		Config_Data.CW_FF:=0;
	
	1:
		Temp_C:=TO_INT(Unit_Convert(eFrom:=Temperature_Units,eTo:=eUnits.C,Source:=Combined_Temp.EU));
		Flow_LPM:=TO_INT(Unit_Convert(eFrom:=Flow_Units,eTo:=eUnits.lpm,Source:=Config_Data.Flow_Rate));
		Config_Data.CW_Base_CV:=	Temp_Flow_CV.Deg_C[Temp_C].lpm[Flow_LPM].CW_CV:=CW_PID.CV;
		Config_Data.HW_Base_CV:= 	Temp_Flow_CV.Deg_C[Temp_C].lpm[Flow_LPM].HW_CV:=HW_PID.CV;
		IF Config_Data.HW_Target_Flow>0 THEN	Config_Data.HW_FF:=LIMIT(0, (Config_data.HW_Base_CV/Config_Data.HW_Target_Flow)*0.75, 20);	END_IF
		IF Config_Data.CW_Target_Flow>0 THEN	Config_Data.CW_FF:=LIMIT(0, (Config_data.CW_Base_CV/Config_Data.CW_Target_Flow)*0.75, 20);	END_IF
		
	2:
		
		
		IF Config_Data.HW_Target_Flow>0 AND Kv_Curve[HW_Target_KV_Index]>0 AND Kv_Curve[HW_Target_KV_Index]<100 THEN
			Config_Data.HW_FF:=LIMIT(0, (Config_data.HW_Base_CV/Config_Data.HW_Target_Flow)*0.50, 20);
		END_IF;
		IF  Config_Data.CW_Target_Flow>0 AND Kv_Curve[CW_Target_KV_Index]>0 AND Kv_Curve[CW_Target_KV_Index]<100 THEN
			Config_Data.CW_FF:=LIMIT(0, (Config_Data.CW_Base_CV/Config_Data.CW_Target_Flow)*0.50, 20);
		END_IF;
		
	3:	IF Config_Data.HW_Target_Flow>0 AND Config_Data.CW_Target_Flow>0 THEN
			Config_data.HW_Base_CV:=	SEL(HW_CV_Mode_3=0,TO_REAL(HW_CV_Mode_3),Config_data.HW_Base_CV);
			Config_Data.CW_Base_CV:=	SEL(CW_CV_Mode_3=0,TO_REAL(CW_CV_Mode_3),Config_data.CW_Base_CV);
			//Config_Data.HW_FF:=LIMIT(0, (Config_data.HW_Base_CV/Config_Data.HW_Target_Flow)*0.750, 20);
			//Config_Data.CW_FF:=LIMIT(0, (Config_Data.CW_Base_CV/Config_Data.CW_Target_Flow)*0.750, 20);
			HW_CV_Ramp(IN:=LIMIT(0, (Config_data.HW_Base_CV/Config_Data.HW_Target_Flow)*0.750, 20),OUT=>Config_Data.HW_FF);
			CW_CV_Ramp(IN:=LIMIT(0, (Config_data.CW_Base_CV/Config_Data.CW_Target_Flow)*0.750, 20),OUT=>Config_Data.CW_FF);
		END_IF;
		
		

END_CASE;

CASE	Config_data.Status.eStatus OF
	eTempered_status.Prime_Start:
		Task_Prime:=FALSE;
		Task_Ton.IN:=FALSE;
		IF Config_Data.HW_Flow_OK AND Config_Data.CW_Flow_OK THEN
			Local_status:=eTempered_Status.Prime_Active;
		END_IF;
	eTempered_Status.Prime_Active:
		Task_Ton.IN:=(Config_Data.HW_Flow_OK AND Config_Data.CW_Flow_OK);
		IF Config_Data.Temperature_OK OR Task_ton.Q THEN
			Local_Status:=eTempered_Status.Prime_Complete;
		END_IF	
	eTempered_status.Prime_Complete:
		Task_Ton.IN:=TRUE;
		Task_Prime:=TRUE;
END_CASE;


IF Config_Data.CW_FF>0 	THEN	CW_PID.FF:=Config_Data.CW_FF; END_IF;
IF Config_Data.HW_FF>0  THEN	HW_PID.FF:=Config_Data.HW_FF; END_IF;
END_METHOD

METHOD Task_Run : BOOL
VAR_INPUT
	Rate:Burkert.cAlarm_Window;
	Temperature:Burkert.cAlarm_Window;
	Volume:REAL;
END_VAR


VAR
	Temp_C:INT;
	Flow_LPM:INT;
	
	
	HW_CV_3:INT;
	CW_CV_3:INT;
	
END_VAR
IF Local_Task<>eTempered_Task.Run THEN
	Local_Task:=eTempered_Task.Run;
	Local_Status:=eTempered_Status.Starting;
	ON_Target:=FALSE;
	Task_Ton.IN:=FALSE;
END_IF;

AUX();
Alarms();
Math();
PID_CTRL();
ACV_CTRL();
Task_Ton();

CASE Config_Data.Mode OF
	eTempered_modes.Mix:		Temperature_PID.PLC_Target:=Temperature.Target;
	eTempered_modes.CW_Only:	
		Temperature_PID.PLC_Target:=CW_Supply_TT.EU;
		Temperature.Target:=CW_Supply_TT.EU;
	eTempered_modes.HW_Only:
		Temperature_PID.PLC_Target:=HW_Supply_TT.EU;
		Temperature.Target:=HW_Supply_TT.EU;
END_CASE;

HW_FIT.Rate.Alarm_Config.Setpoints.Hi_Hi_Alarm	:=Config_Data.HW_Target_Flow+Rate.Alarm_Window;
HW_FIT.Rate.Alarm_Config.Setpoints.Hi_Warn		:=Config_Data.HW_Target_Flow+Rate.Warn_Window;
HW_FIT.Rate.Alarm_Config.Setpoints.Low_Warn		:=Config_Data.HW_Target_Flow-Rate.Warn_Window;
HW_FIT.Rate.Alarm_Config.Setpoints.Low_Low_Alarm		:=Config_Data.HW_Target_Flow-Rate.Alarm_Window;
HW_FIT.Rate.Alarm_Config.Setpoints.Alarm_Debounce			:=Rate.Alarm_Delay;
HW_FIT.Rate.Alarm_Config.Setpoints.Warn_Debounce			:=Rate.Alarm_Delay;


CW_FIT.Rate.Alarm_Config.Setpoints.Hi_Hi_Alarm	:=Config_Data.CW_Target_Flow+Rate.Alarm_Window;
CW_FIT.Rate.Alarm_Config.Setpoints.Hi_Warn		:=Config_Data.CW_Target_Flow+Rate.Warn_Window;
CW_FIT.Rate.Alarm_Config.Setpoints.Low_Warn		:=Config_Data.CW_Target_Flow-Rate.Warn_Window;
CW_FIT.Rate.Alarm_Config.Setpoints.Low_Low_Alarm		:=Config_Data.CW_Target_Flow-Rate.Alarm_Window;
CW_FIT.Rate.Alarm_Config.Setpoints.Alarm_Debounce			:=Rate.Alarm_Delay;
CW_FIT.Rate.Alarm_Config.Setpoints.Warn_Debounce			:=Rate.Alarm_Delay;


Burkert.Alarm_Window_Convert(Window:= Temperature,Config:=Combined_Temp.Alarm_Config);
Combined_temp.Alarm_Config.Setpoints.Alarm_Debounce:=0;
Combined_temp.Alarm_Config.Setpoints.Warn_Debounce:=0;



Config_Data.Status.eStatus:=Status_Test(Local_Status);

Config_Data.Base_Flow:=Rate.Target;


IF Temperature_PID.PLC_Enable THEN
	Config_Data.Target_Temperature:= Temperature_PID.CV;
ELSE
	Config_Data.Target_Temperature:= Temperature_PID.PLC_Target;
END_IF;





//CW_KV_Index:= LIMIT(0,TO_INT(Config_Data.CW_Target_KV*KV_Index_Scalar),100);
//HW_KV_Index:= LIMIT(0,TO_INT(Config_Data.HW_Target_KV*KV_Index_Scalar),100);

IF CW_Target_KV_Index>0 AND Kv_Curve[CW_Target_KV_Index]>0 THEN	Config_Data.CW_Base_CV:=Kv_Curve[CW_Target_KV_Index]; END_IF;
IF HW_Target_KV_Index>0 AND Kv_Curve[HW_Target_KV_Index]>0 THEN	Config_Data.HW_Base_CV:=Kv_Curve[HW_Target_KV_Index]; END_IF;	


IF Config_Data.CW_DP > 5 THEN	CW_CV_Mode_3:=FindClosestIndexSorted(ArrayIn:=CV_2_KV,TargetValue:=Config_Data.CW_Target_KV); END_IF;
IF Config_Data.HW_DP > 5 THEN	HW_CV_Mode_3:=FindClosestIndexSorted(ArrayIn:=CV_2_KV,TargetValue:=Config_Data.HW_Target_KV);	END_IF;
	
CASE Run_mode OF
	
	0:
		CW_PID.FF:=0.0;
		HW_PID.FF:=0.0;
		Config_Data.HW_FF:=0;
		Config_Data.CW_FF:=0;
	
	1:
		Temp_C:=TO_INT(Unit_Convert(eFrom:=Temperature_Units,eTo:=eUnits.C,Source:=Combined_Temp.EU));
		Flow_LPM:=TO_INT(Unit_Convert(eFrom:=Flow_Units,eTo:=eUnits.lpm,Source:=Config_Data.Flow_Rate));
		Config_Data.CW_Base_CV:=	Temp_Flow_CV.Deg_C[Temp_C].lpm[Flow_LPM].CW_CV:=CW_PID.CV;
		Config_Data.HW_Base_CV:= 	Temp_Flow_CV.Deg_C[Temp_C].lpm[Flow_LPM].HW_CV:=HW_PID.CV;
		IF Config_Data.HW_Target_Flow>0 THEN	Config_Data.HW_FF:=LIMIT(0, (Config_data.HW_Base_CV/Config_Data.HW_Target_Flow)*0.75, 20);	END_IF
		IF Config_Data.CW_Target_Flow>0 THEN	Config_Data.CW_FF:=LIMIT(0, (Config_data.CW_Base_CV/Config_Data.CW_Target_Flow)*0.75, 20);	END_IF
		
	2:
		
		
		IF Config_Data.HW_Target_Flow>0 AND Kv_Curve[HW_Target_KV_Index]>0 AND Kv_Curve[HW_Target_KV_Index]<100 THEN
			Config_Data.HW_FF:=LIMIT(0, (Config_data.HW_Base_CV/Config_Data.HW_Target_Flow)*0.50, 20);
		END_IF;
		IF  Config_Data.CW_Target_Flow>0 AND Kv_Curve[CW_Target_KV_Index]>0 AND Kv_Curve[CW_Target_KV_Index]<100 THEN
			Config_Data.CW_FF:=LIMIT(0, (Config_Data.CW_Base_CV/Config_Data.CW_Target_Flow)*0.50, 20);
		END_IF;
		
	3:	IF Config_Data.HW_Target_Flow>0 AND Config_Data.CW_Target_Flow>0 THEN
			Config_data.HW_Base_CV:=	SEL(HW_CV_Mode_3=0,TO_REAL(HW_CV_Mode_3),Config_data.HW_Base_CV);
			HW_CV_Ramp(IN:=LIMIT(0, (Config_data.HW_Base_CV/Config_Data.HW_Target_Flow)*0.750, 20),OUT=>Config_Data.HW_FF);
			//Config_Data.HW_FF:=LIMIT(0, (Config_data.HW_Base_CV/Config_Data.HW_Target_Flow)*0.750, 20);
			//Config_Data.CW_FF:=LIMIT(0, (Config_Data.CW_Base_CV/Config_Data.CW_Target_Flow)*0.750, 20);
		END_IF;
		
		IF Config_Data.CW_Target_Flow>0 THEN
			Config_Data.CW_Base_CV:=	SEL(CW_CV_Mode_3=0,TO_REAL(CW_CV_Mode_3),Config_data.CW_Base_CV);
			CW_CV_Ramp(IN:=LIMIT(0, (Config_data.CW_Base_CV/Config_Data.CW_Target_Flow)*0.750, 20),OUT=>Config_Data.CW_FF);
			//Config_Data.HW_FF:=LIMIT(0, (Config_data.HW_Base_CV/Config_Data.HW_Target_Flow)*0.750, 20);
			//Config_Data.CW_FF:=LIMIT(0, (Config_Data.CW_Base_CV/Config_Data.CW_Target_Flow)*0.750, 20);
		END_IF
		
		

END_CASE;









IF Config_Data.CW_FF>0 	AND Config_data.HW_DP>2 AND Config_data.HW_DP<25 	THEN	CW_PID.FF:=Config_Data.CW_FF; END_IF;
IF Config_Data.HW_FF>0  AND Config_data.CW_DP>2 AND Config_data.CW_DP<25 	THEN	HW_PID.FF:=Config_Data.HW_FF; END_IF;	



CASE	Config_data.Status.eStatus OF
	eTempered_Status.Starting:
		IF Config_Data.Temperature_OK AND Config_Data.HW_Flow_OK AND Config_Data.CW_Flow_OK THEN
			Local_Status:=eTempered_Status.Ready;
			Task_Run:=true;
		Else
			Task_Run:=FALSE;
		END_IF;
	eTempered_Status.Ready:
		Task_Run:=TRUE;
		
END_CASE


IF  Kv_Curve[HW_KV_Index]=0 AND  HW_PID.Err<ABS(0.1) THEN Kv_Curve[HW_KV_Index]:=HW_PID.CV; END_IF;
IF  Kv_Curve[CW_KV_Index]=0 AND  CW_PID.Err<ABS(0.1) THEN Kv_Curve[HW_KV_Index]:=CW_PID.CV; END_IF;
END_METHOD

END_FUNCTION_BLOCK

// 50 Functions/Burkert Library/Alarm_Window_Convert
FUNCTION Alarm_Window_Convert : BOOL
VAR_INPUT
	Window: REFERENCE TO	 Alarm_Window;
	Config:	REFERENCE TO	Burkert.cAlarm_Config;
	
END_VAR
VAR
END_VAR

Config.Debounce:=Window.Alarm_Delay;
Config.Hi_Hi_Alarm:= (Window.Target+Window.Alarm_Window);
Config.Hi_Warn:=(Window.Target+Window.Warn_Window);
Config.Low_warn:=(Window.Target-Window.Warn_Window);
Config.Low_Low_Alarm:=(Window.Target-Window.Alarm_Window);

END_FUNCTION

// Simulators/c8691_CanOpen_Sim
FUNCTION_BLOCK c8691_CanOpen_Sim
VAR_INPUT
	BCV: REFERENCE TO c8691;
END_VAR
VAR_OUTPUT
END_VAR
VAR
END_VAR

BCV.PDO.EndPositions.1:=BCV.PDO.Setpoint.0;
BCV.PDO.EndPositions.0:=NOT(BCV.PDO.Setpoint.0);
BCV.PDO.NamurStatus:=1;

END_FUNCTION_BLOCK

// Simulators/c8694_CanOpen_Sim
FUNCTION c8694_CanOpen_Sim
VAR_INPUT
END_VAR
VAR_OUTPUT
	//CanState:_3SCOS.DED.DEVICE_STATE;
END_VAR
VAR
	//Data:Bytes_Dword;
END_VAR
VAR_IN_OUT
	Device:cCanOpen_8694;
END_VAR


Device.PDO.NamurStatus:=1;

Device.PDO.CMD:=Device.PDO.CMDdigital;
Device.PDO.Pos:=Device.PDO.CMDdigital;

//CanState:=_3SCOS.DED.DEVICE_STATE.RUNNING;


Device.CanOpen.Device_State:=_3SCOS.DED.DEVICE_STATE.RUNNING;

END_FUNCTION

// Simulators/CanOpen_8694_Data_Sim
FUNCTION CanOpen_8694_Data_Sim
VAR_INPUT
END_VAR
VAR_OUTPUT
END_VAR
VAR
	//Data:Bytes_Dword;
END_VAR
VAR_IN_OUT
	Device:cCanOpen_8694;
END_VAR



Device.PDO.NamurStatus:=1;
Device.PDO.Pos:=Device.PDO.CMDdigital;
Device.CanOpen.Device_State:=_3SCOS.DED.DEVICE_STATE.DISABLED;

END_FUNCTION

// Simulators/Contactor_Sim
FUNCTION_BLOCK Contactor_Sim
VAR_INPUT
	Device:Burkert.Contactor_DUT;
END_VAR
VAR_OUTPUT
	FWD_Limit:BOOL;
	Rev_Limit:BOOL;
END_VAR
VAR
	tPos:INT;
	pulse: Burkert_OSCAT_BASIC.CLK_PRG;
END_VAR

Pulse(PT:=T#1S);

IF Pulse.Q THEN
	
	IF Device.Q2 AND tPos>0 THEN tPos:=tPos-1; END_IF;
	IF Device.Q1 AND tPos<100 THEN tPos:=tpos+1; END_IF;
END_IF;


FWD_Limit:=tPos<100;
Rev_Limit:=tPos>0;

END_FUNCTION_BLOCK

// Simulators/Edip_8691_Sim
FUNCTION Edip_8691_Sim
VAR_INPUT
	BCV: Reference to ceDip_8691;;
END_VAR
VAR_OUTPUT
END_VAR
VAR
END_VAR

//BCV.PDO.EndPositions.0:=BCV.PDO.Setpoint.0;
//BCV.PDO.EndPositions.1:=NOT(BCV.PDO.Setpoint.0);
//BCV.PDO.NamurStatus:=1;


(*
Join.tWord[0]:=BCV.RX[0];
BCV.PDO.EndPositions:=Join.tByte[1];

Join.tWord[0]:=BCV.RX[1];
BCV.PDO.NamurStatus:=Join.tByte[1];
Join.tWord[1]:=BCV.RX[2];
Join.tWord[0]:=BCV.RX[3];
BCV.PDO.Position:=Join.tReal;

Join.tByte[0]:=0;
Join.tByte[1]:=BCV.PDO.Setpoint;
BCV.TX:=Join.tWord[0];
*)

//BCV.RX[0].8:=BCV.TX.8;
//BCV.RX[0].9:=NOT(BCV.TX.8);
//BCV.RX[1]:=256;

END_FUNCTION

// Simulators/Edip_8694_Data_Sim
FUNCTION Edip_8694_Data_Sim
VAR_INPUT
END_VAR
VAR_OUTPUT
END_VAR
VAR
	//Data:Bytes_Dword;
END_VAR
VAR_IN_OUT
	Device:ceDip_8694;
END_VAR


Device.RX.ActualPosition.tWord[0]:=Device.TX_CmdDigital.tWord[0];
Device.RX.ActualPosition.tWord[1]:=Device.TX_CmdDigital.tWord[1];

Device.RX.NamurStatus.tByte[1]:=1;

Device.RX.CurrentSetPoint.tWord[0]:=Device.TX_CmdDigital.tWord[0];
Device.RX.CurrentSetPoint.tWord[1]:=Device.TX_CmdDigital.tWord[1];


//Device.RX[5]:=0;

END_FUNCTION

// Simulators/eDip_ME44_DI_Count_Sim
FUNCTION eDip_ME44_DI_Count_Sim : Bool
VAR_INPUT
	Pulse_250:BOOL;
	Rate_LPM:REAL;
	FIT:Burkert.cFIT;
	//Current:REAL;
	
END_VAR
VAR
	//Data:Bytes_Dword;
END_VAR

VAR_OUTPUT
	Count:REAL;
END_VAR



IF NOT(FIT.PLC_Reset) AND NOT(FIT.HMI_Reset) THEN
	IF Pulse_250 THEN
		Count:=FIT.Counts+(((Rate_LPM/60)/4)*FIT.K);
	ELSE
		Count:=FIT.Counts;
	END_IF;
ELSE
	Count:=0;	
END_IF;

END_FUNCTION

// Simulators/eDip_ME44_DI_Hz_Sim
FUNCTION eDip_ME44_DI_Hz_Sim : Bool
VAR_INPUT

	Rate_LPM:REAL;
	FIT:Burkert.cFIT;
	
END_VAR
VAR
	//Data:Bytes_Dword;
	//Value:REAL;
END_VAR

VAR_OUTPUT
	Hz:Real;
END_VAR

IF NOT(FIT.PLC_Reset) AND NOT(FIT.HMI_Reset) THEN
	Hz:=(Rate_LPM/60)*FIT.K;
ELSE
	Hz:=0;	
END_IF;

END_FUNCTION

// Simulators/FIT_Sim
FUNCTION FIT_Sim : UDINT
VAR_INPUT
	FIT: REFERENCE TO Burkert.cFIT;
	Control:REAL;
	clk:Bool;
	
END_VAR
VAR_OUTPUT
	Hz:REAL;
END_VAR
VAR
	PLC_Time:UDINT;
END_VAR

IF FIT.HMI_Reset OR FIT.PLC_Reset THEN
	FIT.Counts:=0;
END_IF;

IF clk THEN	
	FIT.Counts:=(FIT.Counts + TO_UDINT(Control/4) );
	IF FIT.Counts=0 THEN FIT.Counts:=1; END_IF;
	
	
END_IF;
FIT_Sim:=FIT.Counts;
Hz:=(Control);

END_FUNCTION

// Simulators/Mix_Sim
FUNCTION Mix_Sim : REAL;
VAR_INPUT
	HW:REAL;
	CW:REAL;
	Temp:REAL;
	RAW_Scale:Burkert.cAnalog_Scale;
END_VAR
VAR
	
END_VAR
VAR_OUTPUT
	Target_Temp:REAL;
END_VAR

	IF HW<>CW then
		Target_temp:=Burkert_OSCAT_BASIC.SCALE_R(
		X:= ((HW-CW)/(HW+CW)), 
		I_LO:= (-1), 
		I_HI:= 1, 
		O_LO:= 0, 
		O_HI:= Temp);
	ELSE
		Target_Temp:=Temp/2;
	END_IF;
	
	Mix_Sim:=Burkert_OSCAT_BASIC.SCALE_R(
	X:= Target_Temp, 
	I_LO:= Raw_Scale.Eu_Min, 
	I_HI:= Raw_Scale.Eu_Max, 
	O_LO:= Raw_Scale.Raw_Min, 
	O_HI:= Raw_Scale.Raw_Max);

END_FUNCTION

// Simulators/TT_SIM
FUNCTION TT_SIM : Bool
VAR_INPUT
	TT: REFERENCE TO Burkert.cAIT;
	Rate_Up:REAL;
	Rate_Down:REAL;
END_VAR
VAR
END_VAR

TT.Analog_Scale.Raw:=TT.Analog_Scale.Raw+(Rate_up-Rate_Down);
TT.Analog_Scale.Raw:=LIMIT(TT.Analog_Scale.Raw_Min,TT.Analog_Scale.Raw,TT.Analog_Scale.Raw_Max);

END_FUNCTION

// Simulators/Vacon_VFD_SIM
FUNCTION_BLOCK Vacon_VFD_SIM
VAR_INPUT
	Device:VFD_Vacon_DUT;
END_VAR
VAR_OUTPUT
END_VAR
VAR
	//Random:REAL;
END_VAR
VAR_IN_OUT
	mbTCP:Vacon_MbTCP;
END_VAR

//Random:=Burkert_OSCAT_BASIC.RDM(Random);
mbTCP.RX[9]:=691;
mbTCP.rx[0].1:=FALSE;// Running Bit
mbTCP.rx[0].2:=TRUE;//FWD BIT;
CASE Device.MODE.eMode	 OF
		eVFD_Modes.Auto:	IF Device.PLC_Run THEN
					mbTCP.RX[0]:=35;
					mbTCP.rx[0].1:=TRUE;
					mbTCP.rx[0].2:=(Device.PLC_CMD>0);
					mbTCP.RX[3]:=REAL_TO_WORD(ABS(Device.PLC_CMD)*6);
				ELSE
					mbTCP.RX[0]:=1;
					mbTCP.RX[3]:=0;
				END_IF;
		eVFD_Modes.Disabled:	mbTCP.RX[0]:=1;
			mbTCP.RX[3]:=0;
		eVFD_Modes.Manual:	mbTCP.RX[0]:=35;
			mbTCP.rx[0].1:=TRUE;
			mbTCP.rx[0].2:=(Device.PLC_CMD>0);
			mbTCP.RX[3]:=REAL_TO_WORD(ABS(Device.MAN_CMD) *6);
END_CASE

END_FUNCTION_BLOCK

// AC2916
FUNCTION_BLOCK AC2916
VAR_INPUT
	CH1:Asi_node_DUT;
	CH2:ASI_Node_DUT;
END_VAR
VAR_OUTPUT
	AC2916:AC2916_DUT;
END_VAR
VAR
END_VAR

AC2916.AI[1] := Ch1.Analog_RX_0;
AC2916.AI[2] := Ch1.Analog_RX_1;
AC2916.AI[3] := Ch2.Analog_RX_0;
AC2916.AI[4] := Ch2.Analog_RX_1;
AC2916.Active := CH1.Active;
Ac2916.Detected := CH1.Detected;
AC2916.PROJECTED := CH1.PROJECTED;
AC2916.Fault := Ch1.Fault;

END_FUNCTION_BLOCK

// Asi_GW_FUN
FUNCTION_BLOCK Asi_GW_FUN
VAR_INPUT
	Flags:ARRAY[0..7] OF DWORD;
	Analog_1_RX:ARRAY[0..79] OF WORD;
	Analog_2_RX:ARRAY[0..74] OF WORD;
	Digital_RX:ARRAY[0..63] OF BYTE;
	
END_VAR
VAR_OUTPUT
	Analog_1_TX:ARRAY[0..79] OF WORD;
	Analog_2_TX:ARRAY[0..74] OF WORD;
	Digital_TX:ARRAY[0..63] OF BYTE;
END_VAR
VAR
	index:INT:=0;
	Offset:INT;
END_VAR

VAR_IN_OUT
	A_Nodes:ARRAY[1..32] OF Asi_node_DUT;
	B_Nodes:ARRAY[1..32] OF Asi_Node_Dut;
END_VAR

FOR index:=1 TO 32 BY 1 DO
	
	A_Nodes[Index].Active:=GETBIT(X:=flags[0] , N:=TO_BYTE(Index) );
	B_Nodes[Index].Active:=GETBIT(X:=flags[1] , N:=TO_BYTE(Index) );
	
	A_Nodes[Index].Detected:=GETBIT(X:=flags[2] , N:=TO_BYTE(Index) );
	B_Nodes[Index].Detected:=GETBIT(X:=flags[3] , N:=TO_BYTE(Index) );
	
	A_Nodes[Index].Fault:=GETBIT(X:=flags[4] , N:=TO_BYTE(Index) );
	B_Nodes[Index].Fault:=GETBIT(X:=flags[5] , N:=TO_BYTE(Index) );
	
	A_Nodes[Index].PROJECTED:=GETBIT(X:=flags[6] , N:=TO_BYTE(Index) );
	B_Nodes[Index].PROJECTED:=GETBIT(X:=flags[7] , N:=TO_BYTE(Index) );
	

	A_Nodes[Index].Digital_RX:=Digital_RX[(Index-1)];
	B_Nodes[Index].Digital_RX:=Digital_RX[(Index+31)];
	
	Digital_TX[Index-1]:=A_Nodes[Index].Digital_TX;
	Digital_TX[Index+31]:=B_Nodes[Index].Digital_TX;
	
	
	IF Index < 17 THEN
		Offset := ((Index-1)*5);
		A_Nodes[Index].Analog_RX_0:=Analog_1_RX[Offset];
		A_Nodes[Index].Analog_RX_1:=Analog_1_RX[Offset+1];
		B_Nodes[Index].Analog_RX_0:=Analog_1_RX[Offset+2];
		B_Nodes[Index].Analog_RX_1:=Analog_1_RX[Offset+3];
		
		Analog_1_TX[Offset]:=A_Nodes[Index].Analog_TX_0;
		Analog_1_TX[Offset+1]:=A_Nodes[Index].Analog_TX_1;
		Analog_1_TX[Offset+2]:=B_Nodes[Index].Analog_TX_0;
		Analog_1_TX[Offset+3]:=B_Nodes[Index].Analog_TX_1;
		
		
	ELSE
		Offset := ((Index-17)*5);
		A_Nodes[Index].Analog_RX_0:=Analog_2_RX[Offset];
		A_Nodes[Index].Analog_RX_1:=Analog_2_RX[Offset+1];
		B_Nodes[Index].Analog_RX_0:=Analog_2_RX[Offset+2];
		B_Nodes[Index].Analog_RX_1:=Analog_2_RX[Offset+3];
		
		Analog_2_TX[Offset]:=A_Nodes[Index].Analog_TX_0;
		Analog_2_TX[Offset+1]:=A_Nodes[Index].Analog_TX_1;
		Analog_2_TX[Offset+2]:=B_Nodes[Index].Analog_TX_0;
		Analog_2_TX[Offset+3]:=B_Nodes[Index].Analog_TX_1;
		
	END_IF;
	
	
END_FOR;

END_FUNCTION_BLOCK

// 50 Functions/Burkert Library/ASi_8694_Mapping
FUNCTION ASi_8694_Mapping : BOOL
VAR_INPUT
	Data_In:WORD;
	Setpoint:REAL;
END_VAR
VAR
END_VAR
VAR_OUTPUT
	Actual:REAL;
	Data_Out:word;
END_VAR

Actual := (INT_TO_REAL(WORD_TO_INT(Data_In))) / 100.0;
Data_Out := REAL_TO_WORD(Setpoint * 100.0);

END_FUNCTION

// 50 Functions/Burkert Library/b8619_CND_FB
FUNCTION_BLOCK b8619_CND_FB
VAR_INPUT
	RX:POINTER TO BYTE;
END_VAR
VAR_OUTPUT
	Data:B8619_CND_DUT;
END_VAR
VAR
	Raw_ID:BYTE;
	Raw_Status:Byte;
END_VAR

raw_id:=rx[0];
	data.ID_Revision.0:=Raw_ID.0;
	data.ID_Revision.1:=Raw_id.1;
	Data.ID_Revision.2:=Raw_id.2;
	Data.ID_Revision.3:=Raw_id.3;
	
	Data.ID_Version.0:=Raw_id.4;
	Data.ID_Version.1:=Raw_ID.5;
	Data.ID_Version.2:=Raw_ID.6;
	Data.ID_Version.3:=Raw_ID.7;
raw_id:=rx[1];
	Data.ID_Slot.0:=Raw_ID.0;
	Data.ID_Slot.1:=Raw_ID.1;
	Data.ID_Slot.2:=Raw_ID.2;
	Data.ID_Slot.3:=Raw_ID.3;
	
	Data.ID_Type.0:=Raw_ID.4;
	Data.ID_Type.1:=Raw_ID.5;
	Data.ID_Type.2:=Raw_ID.6;
	Data.ID_Type.3:=Raw_ID.7;
	
Raw_Status:=RX[2];
	Data.Status_Link_Lost:=Raw_Status.0;
	Data.Status_Calibration_Lost:=Raw_Status.1;
	Data.Status_UserData_lost:=Raw_Status.2;
	Data.Status_Factory_Data_Lost:=Raw_Status.3;
	Data.Status_Probe_Error:=Raw_Status.4;
	Data.Status_Probe_Warning:=Raw_Status.6;
Raw_Status:=RX[3];
	Data.Status_Probe_Calibration	:=Raw_Status.0;
	Data.Status_Presence:=Raw_Status.7;

MEMUtils.MemCpy(pbyDest:=ADR(Data.Temp_Status) , pbySrc:=rx+4 , dwSize:=2 );
MEMUtils.MemCpy(pbyDest:=ADR(Data.CND_Status) , pbySrc:=rx+6 , dwSize:=2 );
MEMUtils.MemCpy(pbyDest:=ADR(Data.RTD)+2 , pbySrc:=rx+12 , dwSize:=2 );
MEMUtils.MemCpy(pbyDest:=ADR(Data.RTD) , pbySrc:=rx+14 , dwSize:=2 );

MEMUtils.MemCpy(pbyDest:=ADR(Data.Temperature)+2 , pbySrc:=rx+16 , dwSize:=2 );
MEMUtils.MemCpy(pbyDest:=ADR(Data.Temperature) , pbySrc:=rx+18 , dwSize:=2 );
MEMUtils.MemCpy(pbyDest:=ADR(Data.Conductivity)+2 , pbySrc:=rx+20 , dwSize:=2 );
MEMUtils.MemCpy(pbyDest:=ADR(Data.Conductivity) , pbySrc:=rx+22 , dwSize:=2 );
MEMUtils.MemCpy(pbyDest:=ADR(Data.Resistivity)+2 , pbySrc:=rx+24 , dwSize:=2 );
MEMUtils.MemCpy(pbyDest:=ADR(Data.Resistivity) , pbySrc:=rx+26 , dwSize:=2 );
MEMUtils.MemCpy(pbyDest:=ADR(Data.TDS)+2 , pbySrc:=rx+28 , dwSize:=2 );
MEMUtils.MemCpy(pbyDest:=ADR(Data.TDS) , pbySrc:=rx+30 , dwSize:=2 );
MEMUtils.MemCpy(pbyDest:=ADR(Data.Concentration)+2 , pbySrc:=rx+32 , dwSize:=2 );
MEMUtils.MemCpy(pbyDest:=ADR(Data.Concentration) , pbySrc:=rx+34 , dwSize:=2 );

END_FUNCTION_BLOCK

// 50 Functions/Burkert Library/B8619_Input_FB
FUNCTION_BLOCK B8619_Input_FB
VAR_INPUT
	RX:POINTER TO BYTE;
END_VAR
VAR_OUTPUT
	Data:B8619_inputs_DUT;
END_VAR
VAR
	Raw_ID:BYTE;
	Raw_Status:Byte;
END_VAR

raw_id:=rx[0];
	data.ID_Revision.0:=Raw_ID.0;
	data.ID_Revision.1:=Raw_id.1;
	Data.ID_Revision.2:=Raw_id.2;
	Data.ID_Revision.3:=Raw_id.3;
	
	Data.ID_Version.0:=Raw_id.4;
	Data.ID_Version.1:=Raw_ID.5;
	Data.ID_Version.2:=Raw_ID.6;
	Data.ID_Version.3:=Raw_ID.7;
raw_id:=rx[1];
	Data.ID_Slot.0:=Raw_ID.0;
	Data.ID_Slot.1:=Raw_ID.1;
	Data.ID_Slot.2:=Raw_ID.2;
	Data.ID_Slot.3:=Raw_ID.3;
	
	Data.ID_Type.0:=Raw_ID.4;
	Data.ID_Type.1:=Raw_ID.5;
	Data.ID_Type.2:=Raw_ID.6;
	Data.ID_Type.3:=Raw_ID.7;
	
Raw_Status:=RX[2];
	Data.Status_Link_Lost:=Raw_Status.0;
	Data.Status_Calibration_Lost:=Raw_Status.1;
	Data.Status_UserData_lost:=Raw_Status.2;
	Data.Status_Factory_Data_Lost:=Raw_Status.3;
	Data.Status_time_lost:=Raw_Status.4;
	Data.Status_Warning:=Raw_Status.6;
Raw_Status:=RX[3];
	Data.Status_Memory_Issue	:=Raw_Status.0;
	Data.Status_Presence:=Raw_Status.7;
	

MEMUtils.MemCpy(pbyDest:=ADR(Data.DI1_Status) , pbySrc:=rx+4 , dwSize:=2);
MEMUtils.MemCpy(pbyDest:=ADR(Data.DI2_Status) , pbySrc:=rx+6 , dwSize:=2);
MEMUtils.MemCpy(pbyDest:=ADR(Data.AI1_Status) , pbySrc:=rx+8 , dwSize:=2);
MEMUtils.MemCpy(pbyDest:=ADR(Data.AI2_Status) , pbySrc:=rx+10 , dwSize:=2);

MEMUtils.MemCpy(pbyDest:=ADR(Data.DI1_Hz)+2 , pbySrc:=rx+12 , dwSize:=2);
MEMUtils.MemCpy(pbyDest:=ADR(Data.DI1_Hz) , pbySrc:=rx+14 , dwSize:=2);

MEMUtils.MemCpy(pbyDest:=ADR(Data.DI1_Flow)+2 , pbySrc:=rx+16 , dwSize:=2);
MEMUtils.MemCpy(pbyDest:=ADR(Data.DI1_Flow) , pbySrc:=rx+18 , dwSize:=2);

MEMUtils.MemCpy(pbyDest:=ADR(Data.DI1_Total_A)+2 , pbySrc:=rx+20 , dwSize:=2);
MEMUtils.MemCpy(pbyDest:=ADR(Data.DI1_Total_A) , pbySrc:=rx+22 , dwSize:=2);

MEMUtils.MemCpy(pbyDest:=ADR(Data.DI1_Total_B)+2 , pbySrc:=rx+24 , dwSize:=2);
MEMUtils.MemCpy(pbyDest:=ADR(Data.DI1_Total_B) , pbySrc:=rx+26 , dwSize:=2);	

MEMUtils.MemCpy(pbyDest:=ADR(Data.DI2_Hz)+2 , pbySrc:=rx+28 , dwSize:=2);
MEMUtils.MemCpy(pbyDest:=ADR(Data.DI2_Hz) , pbySrc:=rx+30 , dwSize:=2);

MEMUtils.MemCpy(pbyDest:=ADR(Data.DI2_Flow)+2 , pbySrc:=rx+32 , dwSize:=2);
MEMUtils.MemCpy(pbyDest:=ADR(Data.DI2_Flow) , pbySrc:=rx+34 , dwSize:=2);

MEMUtils.MemCpy(pbyDest:=ADR(Data.DI2_Total_A)+2 , pbySrc:=rx+36 , dwSize:=2);
MEMUtils.MemCpy(pbyDest:=ADR(Data.DI2_Total_A) , pbySrc:=rx+38 , dwSize:=2);

MEMUtils.MemCpy(pbyDest:=ADR(Data.DI2_Total_B)+2 , pbySrc:=rx+40 , dwSize:=2);
MEMUtils.MemCpy(pbyDest:=ADR(Data.DI2_Total_B) , pbySrc:=rx+42 , dwSize:=2);	

MEMUtils.MemCpy(pbyDest:=ADR(Data.AI1_Raw)+2 , pbySrc:=rx+44 , dwSize:=2);
MEMUtils.MemCpy(pbyDest:=ADR(Data.AI1_Raw) , pbySrc:=rx+46 , dwSize:=2);

MEMUtils.MemCpy(pbyDest:=ADR(Data.AI1_EU)+2 , pbySrc:=rx+48 , dwSize:=2);
MEMUtils.MemCpy(pbyDest:=ADR(Data.AI1_EU) , pbySrc:=rx+50 , dwSize:=2);

MEMUtils.MemCpy(pbyDest:=ADR(Data.AI2_Raw)+2 , pbySrc:=rx+52 , dwSize:=2);
MEMUtils.MemCpy(pbyDest:=ADR(Data.AI2_Raw) , pbySrc:=rx+54 , dwSize:=2);

MEMUtils.MemCpy(pbyDest:=ADR(Data.AI2_EU)+2 , pbySrc:=rx+56 , dwSize:=2);
MEMUtils.MemCpy(pbyDest:=ADR(Data.AI2_EU) , pbySrc:=rx+58 , dwSize:=2);

END_FUNCTION_BLOCK

// 50 Functions/Burkert Library/B8619_Main_FB
FUNCTION_BLOCK B8619_Main_FB
VAR_INPUT
	RX:POINTER TO BYTE;
END_VAR
VAR_OUTPUT
	Data:B8619_Main_DUT;
END_VAR
VAR
	Raw_ID:BYTE;
	Raw_Status:Byte;
END_VAR

raw_id:=rx[0];
	data.ID_Revision.0:=Raw_ID.0;
	data.ID_Revision.1:=Raw_id.1;
	Data.ID_Revision.2:=Raw_id.2;
	Data.ID_Revision.3:=Raw_id.3;
	
	Data.ID_Version.0:=Raw_id.4;
	Data.ID_Version.1:=Raw_ID.5;
	Data.ID_Version.2:=Raw_ID.6;
	Data.ID_Version.3:=Raw_ID.7;
raw_id:=rx[1];
	Data.ID_Slot.0:=Raw_ID.0;
	Data.ID_Slot.1:=Raw_ID.1;
	Data.ID_Slot.2:=Raw_ID.2;
	Data.ID_Slot.3:=Raw_ID.3;
	
	Data.ID_Type.0:=Raw_ID.4;
	Data.ID_Type.1:=Raw_ID.5;
	Data.ID_Type.2:=Raw_ID.6;
	Data.ID_Type.3:=Raw_ID.7;
	
Raw_Status:=RX[2];
	Data.Status_Link_Lost:=Raw_Status.0;
	Data.Status_Calibration_Lost:=Raw_Status.1;
	Data.Status_UserData_lost:=Raw_Status.2;
	Data.Status_Factory_Data_Lost:=Raw_Status.3;
	Data.Status_time_lost:=Raw_Status.4;
	Data.Status_Warning:=Raw_Status.6;
Raw_Status:=RX[3];
	Data.Status_Memory_Issue	:=Raw_Status.0;
	Data.Status_Presence:=Raw_Status.7;
	
MEMUtils.MemCpy(pbyDest:=ADR(Data.M1_M3_Status) , pbySrc:=rx+4 , dwSize:=2 );
MEMUtils.MemCpy(pbyDest:=ADR(Data.M4_M6_Status) , pbySrc:=rx+6 , dwSize:=2);
MEMUtils.MemCpy(pbyDest:=ADR(Data.System_Switch) , pbySrc:=rx+8 , dwSize:=2);
MEMUtils.MemCpy(pbyDest:=ADR(Data.DI1_Status) , pbySrc:=rx+10 , dwSize:=2);
MEMUtils.MemCpy(pbyDest:=ADR(Data.DI2_Status) , pbySrc:=rx+12 , dwSize:=2);
MEMUtils.MemCpy(pbyDest:=ADR(Data.DO1) , pbySrc:=rx+14 , dwSize:=2);
MEMUtils.MemCpy(pbyDest:=ADR(Data.DO2) , pbySrc:=rx+16 , dwSize:=2);

MEMUtils.MemCpy(pbyDest:=ADR(Data.AO1) , pbySrc:=rx+18 , dwSize:=2);
MEMUtils.MemCpy(pbyDest:=ADR(Data.AO1)+2 , pbySrc:=rx+20 , dwSize:=2);

MEMUtils.MemCpy(pbyDest:=ADR(Data.AO2) , pbySrc:=rx+22 , dwSize:=2);
MEMUtils.MemCpy(pbyDest:=ADR(Data.AO2)+2 , pbySrc:=rx+24 , dwSize:=2);

MEMUtils.MemCpy(pbyDest:=ADR(Data.DI1_Hz) , pbySrc:=rx+26 , dwSize:=2);
MEMUtils.MemCpy(pbyDest:=ADR(Data.DI1_Hz)+2 , pbySrc:=rx+28 , dwSize:=2);

MEMUtils.MemCpy(pbyDest:=ADR(Data.DI1_Flow) , pbySrc:=rx+30 , dwSize:=2);
MEMUtils.MemCpy(pbyDest:=ADR(Data.DI1_Flow)+2 , pbySrc:=rx+32 , dwSize:=2);

MEMUtils.MemCpy(pbyDest:=ADR(Data.DI1_Total_A) , pbySrc:=rx+34 , dwSize:=2);
MEMUtils.MemCpy(pbyDest:=ADR(Data.DI1_Total_A)+2 , pbySrc:=rx+36 , dwSize:=2);

MEMUtils.MemCpy(pbyDest:=ADR(Data.DI1_Total_B) , pbySrc:=rx+38 , dwSize:=2);
MEMUtils.MemCpy(pbyDest:=ADR(Data.DI1_Total_B)+2 , pbySrc:=rx+40 , dwSize:=2);	

MEMUtils.MemCpy(pbyDest:=ADR(Data.DI2_Hz) , pbySrc:=rx+42 , dwSize:=2);
MEMUtils.MemCpy(pbyDest:=ADR(Data.DI2_Hz)+2 , pbySrc:=rx+44 , dwSize:=2);

MEMUtils.MemCpy(pbyDest:=ADR(Data.DI2_Flow) , pbySrc:=rx+46 , dwSize:=2);
MEMUtils.MemCpy(pbyDest:=ADR(Data.DI2_Flow)+2 , pbySrc:=rx+48 , dwSize:=2);

MEMUtils.MemCpy(pbyDest:=ADR(Data.DI2_Total_A) , pbySrc:=rx+50 , dwSize:=2);
MEMUtils.MemCpy(pbyDest:=ADR(Data.DI2_Total_A)+2 , pbySrc:=rx+52 , dwSize:=2);

MEMUtils.MemCpy(pbyDest:=ADR(Data.DI2_Total_B) , pbySrc:=rx+54 , dwSize:=2);
MEMUtils.MemCpy(pbyDest:=ADR(Data.DI2_Total_B)+2 , pbySrc:=rx+56 , dwSize:=2);

END_FUNCTION_BLOCK

// 50 Functions/Burkert Library/b8619_PH_ORP_FB
FUNCTION_BLOCK b8619_PH_ORP_FB
VAR_INPUT
	RX:POINTER TO BYTE;
END_VAR
VAR_OUTPUT
	Data:B8619_PH_DUT;
END_VAR
VAR
	Raw_ID:BYTE;
	Raw_Status:Byte;
END_VAR

raw_id:=rx[0];
	data.ID_Revision.0:=Raw_ID.0;
	data.ID_Revision.1:=Raw_id.1;
	Data.ID_Revision.2:=Raw_id.2;
	Data.ID_Revision.3:=Raw_id.3;
	
	Data.ID_Version.0:=Raw_id.4;
	Data.ID_Version.1:=Raw_ID.5;
	Data.ID_Version.2:=Raw_ID.6;
	Data.ID_Version.3:=Raw_ID.7;
raw_id:=rx[1];
	Data.ID_Slot.0:=Raw_ID.0;
	Data.ID_Slot.1:=Raw_ID.1;
	Data.ID_Slot.2:=Raw_ID.2;
	Data.ID_Slot.3:=Raw_ID.3;
	
	Data.ID_Type.0:=Raw_ID.4;
	Data.ID_Type.1:=Raw_ID.5;
	Data.ID_Type.2:=Raw_ID.6;
	Data.ID_Type.3:=Raw_ID.7;
	
Raw_Status:=RX[2];
	Data.Status_Link_Lost:=Raw_Status.0;
	Data.Status_Calibration_Lost:=Raw_Status.1;
	Data.Status_UserData_lost:=Raw_Status.2;
	Data.Status_Factory_Data_Lost:=Raw_Status.3;
	Data.Status_Probe_Error:=Raw_Status.4;
	Data.Status_Probe_Warning:=Raw_Status.6;
Raw_Status:=RX[3];
	Data.Status_Probe_Calibration	:=Raw_Status.0;
	Data.Status_Presence:=Raw_Status.7;

MEMUtils.MemCpy(pbyDest:=ADR(Data.Temp_Status) , pbySrc:=ADR(rx)+4 , dwSize:=2 );
MEMUtils.MemCpy(pbyDest:=ADR(Data.PH_Status) , pbySrc:=ADR(rx)+6 , dwSize:=2 );
MEMUtils.MemCpy(pbyDest:=ADR(Data.RTD)+2 , pbySrc:=ADR(rx)+12 , dwSize:=2 );
MEMUtils.MemCpy(pbyDest:=ADR(Data.RTD) , pbySrc:=ADR(rx)+14 , dwSize:=2 );

MEMUtils.MemCpy(pbyDest:=ADR(Data.Temperature)+2 , pbySrc:=ADR(rx)+16 , dwSize:=2 );
MEMUtils.MemCpy(pbyDest:=ADR(Data.Temperature) , pbySrc:=ADR(rx)+18 , dwSize:=2 );
MEMUtils.MemCpy(pbyDest:=ADR(Data.mv_PH)+2 , pbySrc:=ADR(rx)+20 , dwSize:=2 );
MEMUtils.MemCpy(pbyDest:=ADR(Data.mv_PH) , pbySrc:=ADR(rx)+22 , dwSize:=2 );
MEMUtils.MemCpy(pbyDest:=ADR(Data.mv_ORP)+2 , pbySrc:=ADR(rx)+24 , dwSize:=2 );
MEMUtils.MemCpy(pbyDest:=ADR(Data.mv_ORP) , pbySrc:=ADR(rx)+26 , dwSize:=2 );
MEMUtils.MemCpy(pbyDest:=ADR(Data.PH)+2 , pbySrc:=ADR(rx)+28 , dwSize:=2 );
MEMUtils.MemCpy(pbyDest:=ADR(Data.PH) , pbySrc:=ADR(rx)+30 , dwSize:=2 );
MEMUtils.MemCpy(pbyDest:=ADR(Data.Impedance_Glass)+2 , pbySrc:=ADR(rx)+32 , dwSize:=2 );
MEMUtils.MemCpy(pbyDest:=ADR(Data.Impedance_Glass) , pbySrc:=ADR(rx)+34 , dwSize:=2 );
MEMUtils.MemCpy(pbyDest:=ADR(Data.Impedance_Ref)+2 , pbySrc:=ADR(rx)+36 , dwSize:=2 );
MEMUtils.MemCpy(pbyDest:=ADR(Data.Impedance_Ref) , pbySrc:=ADR(rx)+38 , dwSize:=2 );

END_FUNCTION_BLOCK

// 50 Functions/Burkert Library/Build_ORF_Index
FUNCTION Build_ORF_Index : DWORD
VAR_INPUT
	Index:WORD;
	SubIndex:BYTE;
	Node:BYTE;
	Write:BOOL;
END_VAR
VAR
	uORF:Bytes_Dword;
END_VAR

uORF.tWord[0]:=Index;
uORF.tByte[3]:=SubIndex;
IF Write THEN
	uorf.tByte[2]:=node+16#80;
ELSE
	uorf.tByte[2]:=node;
END_IF;

Build_ORF_Index:=uORF.tDword;

END_FUNCTION

// 50 Functions/Burkert Library/FlowWave_Mapping
FUNCTION FlowWave_Mapping : cFLOWave_DUT
VAR_INPUT
	RX:ARRAY[0..17] OF WORD;
END_VAR
VAR
END_VAR

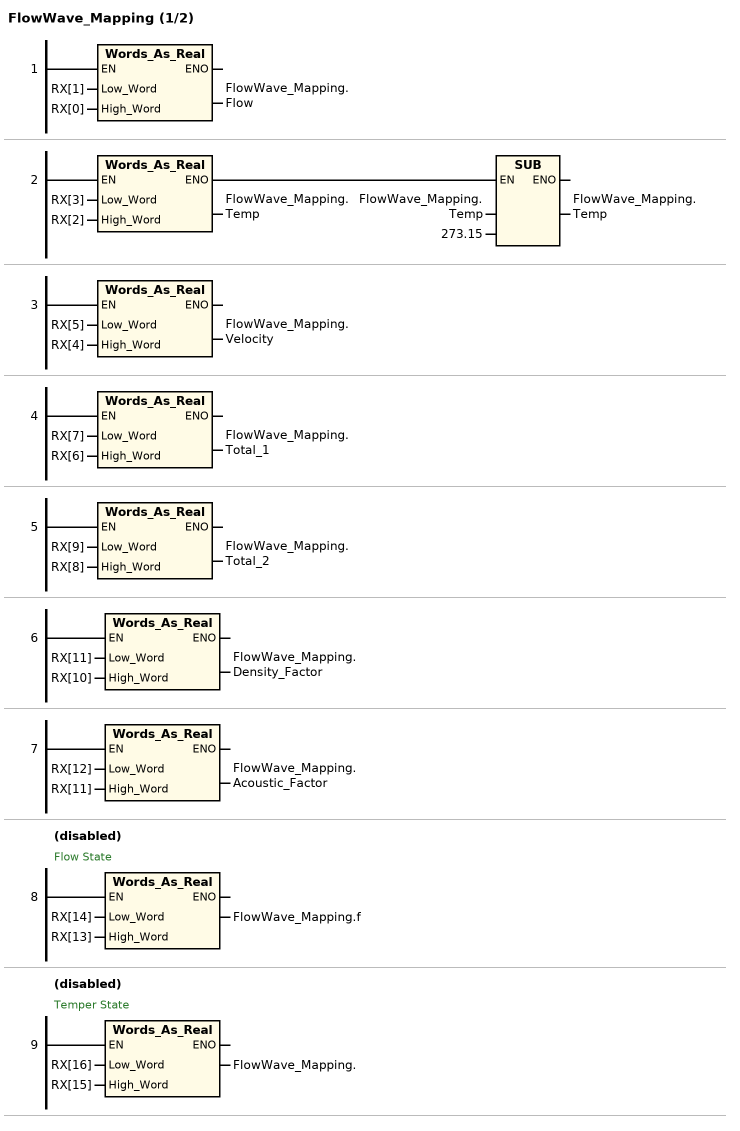
// NETWORK 1
FlowWave_Mapping.Flow := Words_As_Real(Low_Word := RX[1], High_Word := RX[0]);

// NETWORK 2
FlowWave_Mapping.Temp := Words_As_Real(Low_Word := RX[3], High_Word := RX[2]);
FlowWave_Mapping.Temp := FlowWave_Mapping.Temp - 273.15;

// NETWORK 3
FlowWave_Mapping.Velocity := Words_As_Real(Low_Word := RX[5], High_Word := RX[4]);

// NETWORK 4
FlowWave_Mapping.Total_1 := Words_As_Real(Low_Word := RX[7], High_Word := RX[6]);

// NETWORK 5
FlowWave_Mapping.Total_2 := Words_As_Real(Low_Word := RX[9], High_Word := RX[8]);

// NETWORK 6
FlowWave_Mapping.Density_Factor := Words_As_Real(Low_Word := RX[11], High_Word := RX[10]);

// NETWORK 7
FlowWave_Mapping.Acoustic_Factor := Words_As_Real(Low_Word := RX[12], High_Word := RX[11]);

// NETWORK 8 (disabled)
// Flow State
// FlowWave_Mapping.f := Words_As_Real(Low_Word := RX[14], High_Word := RX[13]);

// NETWORK 9 (disabled)
// Temper State
// FlowWave_Mapping. := Words_As_Real(Low_Word := RX[16], High_Word := RX[15]);

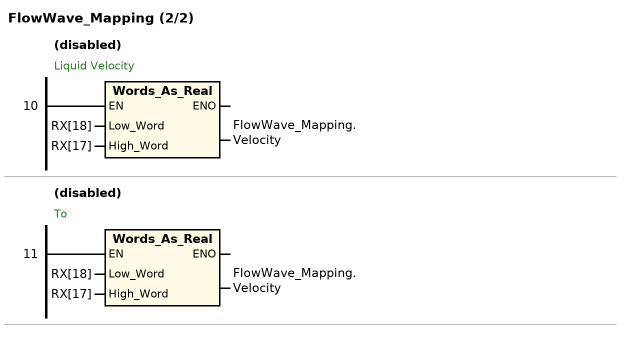
// NETWORK 10 (disabled)
// Liquid Velocity
// FlowWave_Mapping.Velocity := Words_As_Real(Low_Word := RX[18], High_Word := RX[17]);

// NETWORK 11 (disabled)
// To
// FlowWave_Mapping.Velocity := Words_As_Real(Low_Word := RX[18], High_Word := RX[17]);

END_FUNCTION

// 50 Functions/Burkert Library/Tempered_Look_UP
FUNCTION Tempered_Look_UP : Bool
VAR_INPUT
	Data:Tempered_Data;
	
END_VAR

VAR_OUTPUT
	FlowIndex, TempIndex : INT;

	
END_VAR
VAR
	
    FlowIncrement, TempIncrement : REAL;
END_VAR



// Assign values to the increments and target values

// Find the closest indices
FlowIndex := FindClosestIndex(Data.TargetFlow, Data.FlowIncrement, 20);
TempIndex := FindClosestIndex(Data.TargetTemperature, Data.TempIncrement, 20);

// Retrieve the KV values from the array
Data.CW1_KV := Data.Temperature[TempIndex][FlowIndex].CW1_KV;
Data.CW2_KV := Data.Temperature[TempIndex][FlowIndex].CW2_KV;
Data.HW1_KV := Data.Temperature[TempIndex][FlowIndex].HW1_KV;
Data.HW2_KV := Data.Temperature[TempIndex][FlowIndex].HW2_KV;

END_FUNCTION

// f_Fermenter_To_NVL
FUNCTION f_Fermenter_To_NVL : Bool
VAR_INPUT
	LCL:cFermenter_DUT;
END_VAR
VAR_OUTPUT
	NVL:cFermenter_NVL;
END_VAR
VAR
END_VAR

NVL.Crash_Target:=LCL.Crash_Target;

END_FUNCTION

// Burkert Library/Burkert/eDip_ME44_AO
FUNCTION eDip_ME44_AO : bool
VAR_INPUT
	Device: REFERENCE TO cME44_AO;
	
	CH1:REAL;
	CH2:REAL;
	CH3:REAL;
	CH4:REAL;
END_VAR
VAR
	Data:Bytes_Dword;
END_VAR

Device.AO[1]:=Ch1;
Device.AO[2]:=Ch2;
Device.AO[3]:=Ch3;
Device.AO[4]:=Ch4;


Data.tWord[0]:=Device.RX_Namur;
Device.Namur:=Data.tByte[1];

Data.tReal:=Device.AO[1];
Device.TX.CH1[0]:=Data.tWord[0];
Device.TX.CH1[1]:=Data.tWord[1];

Data.tReal:=Device.AO[2];
Device.TX.CH2[0]:=Data.tWord[0];
Device.TX.CH2[1]:=Data.tWord[1];

Data.tReal:=Device.AO[3];
Device.TX.CH3[0]:=Data.tWord[0];
Device.TX.CH3[1]:=Data.tWord[1];

Data.tReal:=Device.AO[4];
Device.TX.CH4[0]:=Data.tWord[0];
Device.TX.CH4[1]:=Data.tWord[1];

END_FUNCTION

// Burkert Library/Burkert/eDip_ME44_DO_Analog
FUNCTION eDip_ME44_DO_Analog : bool
VAR_INPUT
	Device: REFERENCE TO cME44_DO;
	DO_1:BOOL;
	DO_2:BOOL;
	DO_3:BOOL;
	DO_4:BOOL;
	DO_5:BOOL;
	DO_6:BOOL;
	DO_7:BOOL;
	DO_8:BOOL;
	
	PWM_1:REAL;
	PWM_2:REAL;
	PWM_3:REAL;
	PWM_4:REAL;
	PWM_5:REAL;
	PWM_6:REAL;
	PWM_7:REAL;
	PWM_8:REAL;
	
	
	
END_VAR
VAR
	Data:Bytes_Dword;
END_VAR

Data.tWord[0]:=Device.RX_Namur;
Device.Namur:=Data.tByte[1];

Device.TX.CH1Ch8.8:=DO_1;
Device.TX.CH1Ch8.9:=DO_2;
Device.TX.CH1Ch8.10:=DO_3;
Device.TX.CH1Ch8.11:=DO_4;
Device.TX.CH1Ch8.12:=DO_5;
Device.TX.CH1Ch8.13:=DO_6;
Device.TX.CH1Ch8.14:=DO_7;
Device.TX.CH1Ch8.15:=DO_8;


Device.TX.CH1Bin.8:=DO_1;
Device.TX.CH2Bin.8:=DO_2;
Device.TX.CH3Bin.8:=DO_3;
Device.TX.CH4Bin.8:=DO_4;
Device.TX.CH5Bin.8:=DO_5;
Device.TX.CH6Bin.8:=DO_6;
Device.TX.CH7Bin.8:=DO_7;
Device.TX.CH8Bin.8:=DO_8;


Data.tReal:=PWM_1;
Device.TX.CH1Float[0]:=Data.tWord[0];
Device.TX.CH1Float[1]:=Data.tWord[1];

Data.tReal:=PWM_2;
Device.TX.CH2Float[0]:=Data.tWord[0];
Device.TX.CH2Float[1]:=Data.tWord[1];

Data.tReal:=PWM_3;
Device.TX.CH3Float[0]:=Data.tWord[0];
Device.TX.CH3Float[1]:=Data.tWord[1];

Data.tReal:=PWM_4;
Device.TX.CH4Float[0]:=Data.tWord[0];
Device.TX.CH4Float[1]:=Data.tWord[1];

Data.tReal:=PWM_5;
Device.TX.CH5Float[0]:=Data.tWord[0];
Device.TX.CH5Float[1]:=Data.tWord[1];

Data.tReal:=PWM_6;
Device.TX.CH6Float[0]:=Data.tWord[0];
Device.TX.CH6Float[1]:=Data.tWord[1];

Data.tReal:=PWM_7;
Device.TX.CH7Float[0]:=Data.tWord[0];
Device.TX.CH7Float[1]:=Data.tWord[1];

Data.tReal:=PWM_8;
Device.TX.CH8Float[0]:=Data.tWord[0];
Device.TX.CH8Float[1]:=Data.tWord[1];

END_FUNCTION

// Burkert Library/Burkert/eDip_ME44_DO
FUNCTION eDip_ME44_DO : bool
VAR_INPUT
	Device: REFERENCE TO cME44_DO;
	DO_1:BOOL;
	DO_2:BOOL;
	DO_3:BOOL;
	DO_4:BOOL;
	DO_5:BOOL;
	DO_6:BOOL;
	DO_7:BOOL;
	DO_8:BOOL;
	
	
END_VAR
VAR
	Data:Bytes_Dword;
END_VAR

Data.tWord[0]:=Device.RX_Namur;
Device.Namur:=Data.tByte[1];

Device.TX.CH1Ch8.8:=DO_1;
Device.TX.CH1Ch8.9:=DO_2;
Device.TX.CH1Ch8.10:=DO_3;
Device.TX.CH1Ch8.11:=DO_4;
Device.TX.CH1Ch8.12:=DO_5;
Device.TX.CH1Ch8.13:=DO_6;
Device.TX.CH1Ch8.14:=DO_7;
Device.TX.CH1Ch8.15:=DO_8;


Device.TX.CH1Bin.8:=DO_1;
Device.TX.CH2Bin.8:=DO_2;
Device.TX.CH3Bin.8:=DO_3;
Device.TX.CH4Bin.8:=DO_4;
Device.TX.CH5Bin.8:=DO_5;
Device.TX.CH6Bin.8:=DO_6;
Device.TX.CH7Bin.8:=DO_7;
Device.TX.CH8Bin.8:=DO_8;

END_FUNCTION

// Burkert Library/Burkert/eDip_ReadSingleItem
FUNCTION_BLOCK eDip_ReadSingleItem
VAR_INPUT
    Index     : WORD;
    SubIndex  : BYTE;
    Node      : BYTE;
	Enable:BOOL;
	orf:REFERENCE TO eDip_MEx3_ORF;
END_VAR
VAR_OUTPUT
	Data:Bytes_Dword;
	Complete:BOOL;
END_VAR
VAR
	Stage:BYTE:=0;
	Flash:Burkert_OSCAT_BASIC.GEN_PULSE;
	Active_count:UINT:=0;
	Fault_Count:UINT:=0;
	Fault_Code:DWORD;
	Raw_Data:Dword;
	
END_VAR

Flash(ENQ:=TRUE,PTH:=T#50MS,PTL:=T#50MS);

IF NOT(Enable) THEN Stage:=0; END_IF

CASE Stage OF
	0:	Complete:=FALSE;
		Raw_Data:=16#FFFFFFFE;
		IF Enable THEN 
			Stage:=1;
			//ORF.Write_Value:=FALSE;
			END_IF
	1:	//Clear Old Data
		ORF.Call := 0;
        ORF.Length := 16#0400;
        ORF.Value_TX := 16#FFFFFFFF;
		ORF.Index_TX:=Build_Orf_Index(Index:=Index,SubIndex:=SubIndex,Node:=Node,Write:=FALSE);
		ORF.Write_Value:=FALSE;
		Stage:=2;
	2:	ORF.Write_Value:=TRUE;
		Stage:=3;

	3:	ORF.Write_Value:=Flash.Q;
		IF ORF.Index_RX=ORF.Index_TX AND ORF.Value_RX=16#FFFFFFFF	 THEN 
			ORF.Length := 16#0000;
			ORF.Write_Value:=FALSE;
			Orf.Call.8:=TRUE;
			Stage:=6;
		END_IF;
(*
	4: 	Orf.Call.8:=Flash.Q;
		IF Flash.Q THEN Stage:=5; END_IF;
	5: 	IF NOT(Flash.Q) THEN Stage:=6; END_IF;
*)
	6:	Raw_Data:=ORF.Value_RX;
		IF Raw_Data<16#FFFFFFFE	THEN 
			Data.tDword:=MEM.ReverseWORDsInDWORD(dwInput:=Raw_Data );
			Stage:=7; 
		END_IF;
		Orf.Call.8:=TRUE;
		IF ORF.Result=16#FFFFFFFF THEN Active_count:=Active_count+1; END_IF;
		IF ORF.Result>1 AND ORF.Result<16#FFFFFFFF AND Flash.Q	THEN Stage:=9; END_IF;
		
	7:	//First_data:=MEM.ReverseWORDsInDWORD(dwInput:=orf.Value_RX );
		ORF.Value_TX:=0;
		Orf.Call:=16#0000;
		ORF.Write_Value:=FALSE;
		Raw_Data:=16#FFFFFFFD;
		Stage:=8;
	8:	
		Complete:=TRUE;
		ORF.Write_Value:=FALSE;
		Orf.Call:=16#0000;		
	9: 
		Fault_Code:=MEM.ReverseWORDsInDWORD(dwInput:=orf.Result );
		Data.tDword:=0;
		ORF.Index_TX:=Build_Orf_Index(Index:=16#1000,SubIndex:=16#0,Node:=Node,Write:=FALSE);
		Fault_Count:=Fault_Count+1;
		Stage:=10;
	10:
		Orf.Call.8:=Flash.Q;
		IF orf.Result=0 THEN stage:=11;END_IF;
	11:	Orf.Call:=0;
		ORF.Index_TX:=Build_Orf_Index(Index:=Index,SubIndex:=SubIndex,Node:=Node,Write:=FALSE);
		Complete:=TRUE;
END_CASE

END_FUNCTION_BLOCK

// Burkert Library/Burkert/ME43_SDO
FUNCTION_BLOCK ME43_SDO
VAR_INPUT
	CommState:ModbusTCPComState;
	Node:BYTE;
	orf:	REFERENCE TO eDip_MEx3_ORF;
	
	
	r8228:	REFERENCE TO ceDip_8228;
	r8312: 	REFERENCE TO c8312;
	r8412: 	REFERENCE TO c8412;
	r8691:	REFERENCE TO c8691;
	r8694:	REFERENCE TO c8694;
	r8653:	REFERENCE TO c8653;
	rME64:	REFERENCE TO cME64;
	r8098:	REFERENCE TO Burkert.c8098;
	r336x:	REFERENCE TO c336x;
	
	rME44AI:REFERENCE TO cME44_AI;
	
	
END_VAR
VAR_OUTPUT
	Product_Code:DWORD;
	Result:DWORD;
	
END_VAR
VAR
	
Task:eMEx3SDO;
//uORF:Bytes_Dword;
Value:Bytes_Dword;
Pulse:Burkert_OSCAT_BASIC.CLK_PRG;
Active:ARRAY[0..127] OF DWORD;
Scan_Index:UINT;
Device_Stage:UINT;
Scan_Clear_Count:DWORD;

SubStage:BYTE;
Flash:Burkert_OSCAT_BASIC.GEN_PULSE;

ORF_Stage:BYTE:=0;
data:Bytes_Dword;
dio:cDIO;
DSO:cDSO;
DDO:cDDO;


ReadSingleItem:eDip_ReadSingleItem;
WriteSingleItem:eDip_WriteSingleItem;
DirectWriteSingleItem:eDip_WriteSingleItem;
ReadDDO :eDip_ReadDDo;
ReadDSO :eDip_ReadDSO;

Direct_Write_R_trig:R_trig;
t8312:c8312;
t8412:c8412;
t8691:c8691;
t8694:c8694;
t8653:c8653;
t8228:ceDip_8228;
tME44AI:cME44_AI;
tME64:cME64;
t8098:Burkert.c8098;
t336x:c336x;

END_VAR

//0x10180-02 Product Code
orf.CommState:=CommState;
CASE CommState OF
	ModbusTCPComState.OFF: ORF.strTCPstate:='OFF';
	ModbusTCPComState.CONNECTING: ORF.strTCPstate:='CONNECTING';
	ModbusTCPComState.CONNECTED: ORF.strTCPstate:='CONNECTED';
	ModbusTCPComState.DISCONNECTING: ORF.strTCPstate:='DISCONNECTING';
	ModbusTCPComState.SOCKET_ERROR: ORF.strTCPstate:='SOCKET_ERROR';
END_CASE

ReadSingleItem(Node:=Node,orf:=orf);
WriteSingleItem(Node:=Node,orf:=orf);
//DirectWriteSingleItem(Orf:=orf);
ReadDDO(ReadSingleItem:=ReadSingleItem);
ReadDSO(ReadSingleItem:=ReadSingleItem);
Pulse(PT:=T#500MS);
Flash(ENQ:=TRUE,PTH:=T#250MS,PTL:=T#250MS);
Result:=ORF.Value_RX;
Direct_Write_R_trig();
//ORF.Index:=uORF.tDword;

IF Node>127 OR Node=0 OR DirectWriteSingleItem.Enable THEN 
	Task:=eMEx3SDO.Idle;
	ReadSingleItem.Enable:=FALSE;
	WriteSingleItem.Enable:=FALSE;
	product_Code:=0;
	Device_Stage:=0;
	orf.Call:=16#00;
	ORF.Write_Value:=FALSE;
	ReadDDO.Enable:=FALSE;
	ReadDSO.Enable:=FALSE;
ELSE
	IF Product_code=0 OR product_code>16#FFFFFFFA THEN
		ReadSingleItem.Index := 16#1018;
		ReadSingleItem.SubIndex := 16#02;
		ReadSingleItem.Enable:=TRUE;
		IF ReadSingleItem.Complete THEN 
			Product_Code:=ReadSingleItem.Data.tDword;
			ReadSingleItem.Enable:=FALSE;
		END_IF;
	END_IF;
END_IF;


IF ORF.Result=16#FFFFFFFF THEN Orf.Call:=0;END_IF;

CASE product_code OF
	0:		SubStage:=0;Device_Stage:=0;
	8228: 		edip_8228();
	8653: 		edip_8653();
	8691: 		edip_8691();
	8694:		eDip_8694();
	8098:		s8098();
	3363:		eDip_336x();
	1296380980 	:ME44_AI();
	1296381492	:ME64();
		
	
	
END_CASE;


IF Direct_Write_R_trig.CLK AND DirectWriteSingleItem.Enable AND DirectWriteSingleItem.Complete THEN 
	DirectWriteSingleItem.Enable:=FALSE;
	Direct_Write_R_trig.CLK:=FALSE;
END_IF;

METHOD Direct_Write : BOOL
VAR_INPUT
	Node:BYTE;
	Index:WORD;
	SubIndex:BYTE;
	Length:BYTE;
	Data:Dword;
END_VAR
Direct_Write_R_trig.CLK:=TRUE;

DirectWriteSingleItem.Node:=Node;
DirectWriteSingleItem.Index:=Index;
DirectWriteSingleItem.SubIndex:=SubIndex;
DirectWriteSingleItem.Length:=Length;
DirectWriteSingleItem.Data.tDword:=Data;
DirectWriteSingleItem.Enable:=Direct_Write_R_trig.Q;
Direct_Write:=DirectWriteSingleItem.Complete;
END_METHOD

END_FUNCTION_BLOCK

// Level_1_Devices/Burkert Library/eDip/eDip_336x
FUNCTION_BLOCK eDip_336x
VAR_INPUT
	CutOff:REAL;
	LOCKOUT_NC:BOOL;
	Permissive_NC:BOOL;
	Online:BOOL;
	Error_PCT:REAL;
	Error_Delay_S:INT;
	Node:BYTE;
END_VAR
VAR_OUTPUT
END_VAR

VAR
	//Data:Bytes_Dword;
	Base_ACV:Basic_ACV_UDFB;
	//init:BOOL;
END_VAR
VAR_IN_OUT
	Device:ceDip_336x;
END_VAR


PDO_Translate();

Base_ACV.FB:=Device.PDO.Pos;
Base_ACV.CutOff:=CutOff;
Base_ACV.LOCKOUT_NC:=Lockout_NC;
Base_ACV.Online:=Online AND Device.PDO.NamurStatus>0;
Base_ACV.Permissive_NC:=Permissive_NC;
Base_ACV.Error_Delay_S:=Error_Delay_s;
Base_ACV.Error_PCT:=Error_PCT;
Base_ACV(Valve:=Device);

Device.PDO.CMDdigital:=Base_ACV.Output;
Device.DSO.Node:=Node;


(*
CASE Device.PDO.NamurStatus OF
	0:	Device.Status.eStatus:=Burkert.eBCV_Status.OFFLINE;
	2:	Device.Status.eStatus:=Burkert.eBCV_Status.Maintenance_Required;
	3:	Device.Status.eStatus:=Burkert.eBCV_Status.Out_Of_Spec;
	//4:	Device.Status:=Burkert.eBCV_Status.Warning;
	5:	Device.Status.eStatus:=Burkert.eBCV_Status.Error;
	
END_CASE

*)

END_FUNCTION_BLOCK

// Level_1_Devices/Burkert Library/Basic_ACV_UDFB
FUNCTION_BLOCK Basic_ACV_UDFB
VAR_INPUT
	FB:REAL;
	CutOff:REAL;
	LockOut_NC:BOOL;
	Online:BOOL;
	Error_PCT:REAL;
	Error_Delay_S:INT;
	Permissive_NC:BOOL;
END_VAR
VAR_OUTPUT
	Status	:INT;
	Output	:REAL;
END_VAR
VAR_IN_OUT
	Valve	:Burkert.cACV;
END_VAR
VAR
	TON_1: TON;
	TOF_0: TOF;
END_VAR

(* body of a kind this reader does not render *)

END_FUNCTION_BLOCK

// Burkert Library/Burkert/ME44_DI
FUNCTION ME44_DI :BOOL;
VAR_INPUT
		device :REFERENCE TO cME44_DI;
		Node:BYTE;
END_VAR
VAR
	//Data:Bytes_Dword;
END_VAR

Device.DSO.Node:=Node;(*
Device.Namur:=Device.RX.Namur.tByte[1];

Device.Ch[1].Hz_Count:=Device.RX.DI1_Float.tReal;
Device.Ch[2].Hz_Count:=Device.RX.DI2_Float.tReal;
Device.Ch[3].Hz_Count:=Device.RX.DI3_Float.tReal;
Device.Ch[4].Hz_Count:=Device.RX.DI4_Float.tReal;
Device.Ch[5].Hz_Count:=Device.RX.DI5_Float.tReal;
Device.Ch[6].Hz_Count:=Device.RX.DI6_Float.tReal;
Device.Ch[7].Hz_Count:=Device.RX.DI7_Float.tReal;
Device.Ch[8].Hz_Count:=Device.RX.DI8_Float.tReal;

Device.Ch[1].Totaliser:=Device.RX.DI1_Total.tReal;
Device.Ch[2].Totaliser:=Device.RX.DI2_Total.tReal;
Device.Ch[3].Totaliser:=Device.RX.DI3_Total.tReal;
Device.Ch[4].Totaliser:=Device.RX.DI4_Total.tReal;
Device.Ch[5].Totaliser:=Device.RX.DI5_Total.tReal;
Device.Ch[6].Totaliser:=Device.RX.DI6_Total.tReal;
Device.Ch[7].Totaliser:=Device.RX.DI7_Total.tReal;
Device.Ch[8].Totaliser:=Device.RX.DI8_Total.tReal;

Device.Ch[1].Raw:=Device.RX.DI1_DI_8.tByte[1].0;
Device.Ch[2].Raw:=Device.RX.DI1_DI_8.tByte[1].1;
Device.Ch[3].Raw:=Device.RX.DI1_DI_8.tByte[1].2;
Device.Ch[4].Raw:=Device.RX.DI1_DI_8.tByte[1].3;
Device.Ch[5].Raw:=Device.RX.DI1_DI_8.tByte[1].4;
Device.Ch[6].Raw:=Device.RX.DI1_DI_8.tByte[1].5;
Device.Ch[7].Raw:=Device.RX.DI1_DI_8.tByte[1].6;
Device.Ch[8].Raw:=Device.RX.DI1_DI_8.tByte[1].7;





Device.TX.Counter_Reset.8:=Device.Ch[1].Reset_Count;
Device.TX.Totaliser_Reset.8:=Device.Ch[1].Reset_Totaliser;

Device.TX.Counter_Reset.9:=Device.Ch[2].Reset_Count;
Device.TX.Totaliser_Reset.9:=Device.Ch[2].Reset_Totaliser;

Device.TX.Counter_Reset.10:=Device.Ch[3].Reset_Count;
Device.TX.Totaliser_Reset.10:=Device.Ch[3].Reset_Totaliser;

Device.TX.Counter_Reset.11:=Device.Ch[4].Reset_Count;
Device.TX.Totaliser_Reset.11:=Device.Ch[4].Reset_Totaliser;

Device.TX.Counter_Reset.12:=Device.Ch[5].Reset_Count;
Device.TX.Totaliser_Reset.12:=Device.Ch[5].Reset_Totaliser;

Device.TX.Counter_Reset.13:=Device.Ch[6].Reset_Count;
Device.TX.Totaliser_Reset.13:=Device.Ch[6].Reset_Totaliser;

Device.TX.Counter_Reset.14:=Device.Ch[7].Reset_Count;
Device.TX.Totaliser_Reset.14:=Device.Ch[7].Reset_Totaliser;

Device.TX.Counter_Reset.15:=Device.Ch[8].Reset_Count;
Device.TX.Totaliser_Reset.15:=Device.Ch[8].Reset_Totaliser;

*)

END_FUNCTION

// Burkert Library/eDip/eDip_8605_CTRL
FUNCTION_BLOCK eDip_8605_CTRL
VAR_INPUT
	GW_TCP_State:ModbusTCPComState;
	Device: REFERENCE TO ceDip_8605;
	Node:Byte;
END_VAR
VAR_OUTPUT
END_VAR
VAR
	Data:Bytes_Dword;
END_VAR

Parse_RX();
Parse_TX();

Device.DSO.Node:=Node;

CASE GW_TCP_State OF
	ModbusTCPComState.OFF: Device.strTCPstate:='OFF';
	ModbusTCPComState.CONNECTING: Device.strTCPstate:='CONNECTING';
	ModbusTCPComState.CONNECTED: Device.strTCPstate:='CONNECTED';
	ModbusTCPComState.DISCONNECTING: Device.strTCPstate:='DISCONNECTING';
	ModbusTCPComState.SOCKET_ERROR: Device.strTCPstate:='SOCKET_ERROR';
END_CASE

ACTION Parse_TX:
Device.TX.8:=Device.PDO.DO1;
END_ACTION

END_FUNCTION_BLOCK

// Burkert Library/eDip/eDip_ME44_AI
FUNCTION eDip_ME44_AI :BOOL
VAR_INPUT
	Device: REFERENCE TO ceDip_ME44_AI;
	Node:BYTE;
	GW_TCP_State:ModbusTCPComState;
END_VAR
VAR_OUTPUT
END_VAR
VAR
	Data:Bytes_Dword;
END_VAR

Device.DSO.Node:=Node;
Device.Namur.iNamur:=Device.RX.Namur.tByte[1];


Device.AI[1]:=Device.RX.CH1.tReal;

Device.AI[2]:=Device.RX.CH2.tReal;

Device.AI[3]:=Device.RX.CH3.tReal;

Device.AI[4]:=Device.RX.CH4.tReal;

CASE GW_TCP_State OF
	ModbusTCPComState.OFF: Device.strTCPstate:='OFF';
	ModbusTCPComState.CONNECTING: Device.strTCPstate:='CONNECTING';
	ModbusTCPComState.CONNECTED: Device.strTCPstate:='CONNECTED';
	ModbusTCPComState.DISCONNECTING: Device.strTCPstate:='DISCONNECTING';
	ModbusTCPComState.SOCKET_ERROR: Device.strTCPstate:='SOCKET_ERROR';
END_CASE
IF GW_TCP_State<> ModbusTCPComState.CONNECTED THEN
	Device.Namur.eNamur:=eNamur107.Offline;
END_IF;

END_FUNCTION

// Burkert Library/eDip/eDip_ME44_DI
FUNCTION eDip_ME44_DI :BOOL;
VAR_INPUT
		device :REFERENCE TO ceDip_ME44_DI;
		Node:BYTE;
END_VAR
VAR
	//Data:Bytes_Dword;
END_VAR

Device.DSO.Node:=Node;
Device.Namur.iNamur:=Device.RX.Namur.tByte[1];

